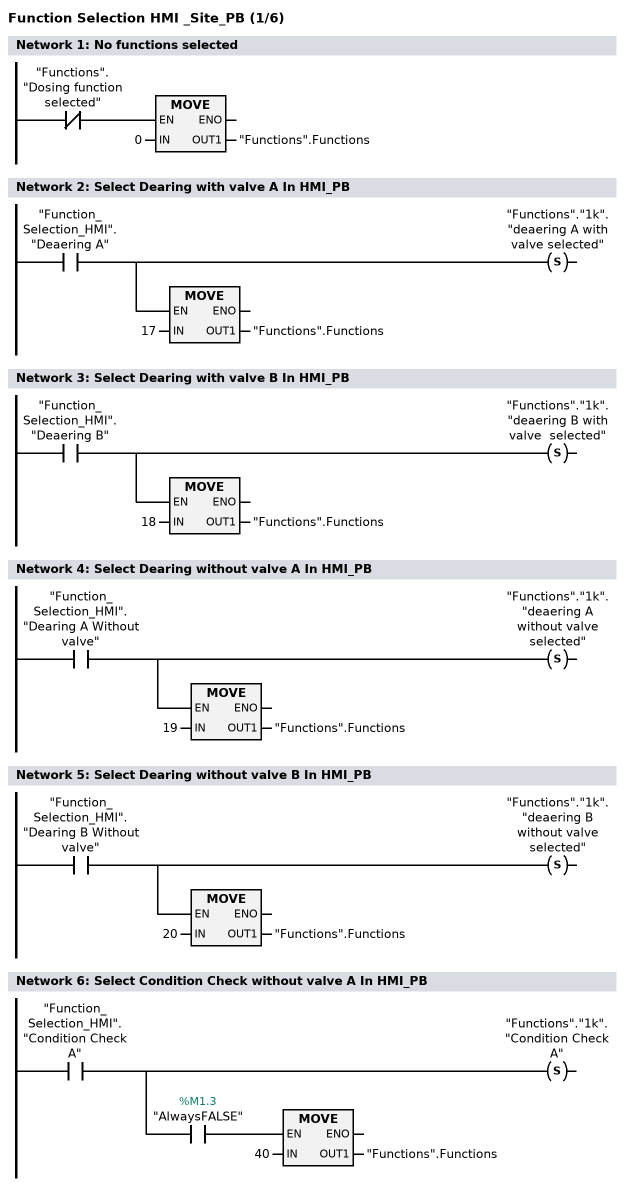
   RUNG wire#powerrail
      I_Contact( "Functions"."Dosing function selected" )
      Move(in := 0, out1 => "Functions".Functions)
   END_RUNG
   // the same network as SCL:
   IF NOT "Functions"."Dosing function selected" THEN "Functions".Functions := 0; END_IF;
END_REGION

REGION Network 2: Select Dearing with valve A In HMI_PB
   RUNG wire#powerrail
      Contact( "Function_Selection_HMI"."Deaering A" )
      wire#w1
      S_Coil( "Functions"."1k"."deaering A with valve selected" )
   END_RUNG
   RUNG wire#w1
      Move(in := 17, out1 => "Functions".Functions)
   END_RUNG
   // the same network as SCL:
   IF "Function_Selection_HMI"."Deaering A" THEN
       "Functions"."1k"."deaering A with valve selected" := TRUE;
       "Functions".Functions := 17;
   END_IF;
END_REGION

REGION Network 3: Select Dearing with valve B In HMI_PB
   RUNG wire#powerrail
      Contact( "Function_Selection_HMI"."Deaering B" )
      wire#w1
      S_Coil( "Functions"."1k"."deaering B with valve  selected" )
   END_RUNG
   RUNG wire#w1
      Move(in := 18, out1 => "Functions".Functions)
   END_RUNG
   // the same network as SCL:
   IF "Function_Selection_HMI"."Deaering B" THEN
       "Functions"."1k"."deaering B with valve  selected" := TRUE;
       "Functions".Functions := 18;
   END_IF;
END_REGION

REGION Network 4: Select Dearing without valve A In HMI_PB
   RUNG wire#powerrail
      Contact( "Function_Selection_HMI"."Dearing A Without valve" )
      wire#w1
      S_Coil( "Functions"."1k"."deaering A without valve selected" )
   END_RUNG
   RUNG wire#w1
      Move(in := 19, out1 => "Functions".Functions)
   END_RUNG
   // the same network as SCL:
   IF "Function_Selection_HMI"."Dearing A Without valve" THEN
       "Functions"."1k"."deaering A without valve selected" := TRUE;
       "Functions".Functions := 19;
   END_IF;
END_REGION

REGION Network 5: Select Dearing without valve B In HMI_PB
   RUNG wire#powerrail
      Contact( "Function_Selection_HMI"."Dearing B Without valve" )
      wire#w1
      S_Coil( "Functions"."1k"."deaering B without valve  selected" )
   END_RUNG
   RUNG wire#w1
      Move(in := 20, out1 => "Functions".Functions)
   END_RUNG
   // the same network as SCL:
   IF "Function_Selection_HMI"."Dearing B Without valve" THEN
       "Functions"."1k"."deaering B without valve  selected" := TRUE;
       "Functions".Functions := 20;
   END_IF;
END_REGION

REGION Network 6: Select Condition Check without valve A In HMI_PB
   RUNG wire#powerrail
      Contact( "Function_Selection_HMI"."Condition Check A" )
      wire#w1
      S_Coil( "Functions"."1k"."Condition Check A" )
   END_RUNG
   RUNG wire#w1
      Contact( "AlwaysFALSE" )
      Move(in := 40, out1 => "Functions".Functions)
   END_RUNG
   // the same network as SCL:
   IF "Function_Selection_HMI"."Condition Check A" THEN "Functions"."1k"."Condition Check A" := TRUE; END_IF;
   IF "Function_Selection_HMI"."Condition Check A" AND "AlwaysFALSE" THEN
       "Functions".Functions := 40;
   END_IF;
END_REGION

REGION Network 7: Select Conditon Check without valve B In HMI_PB
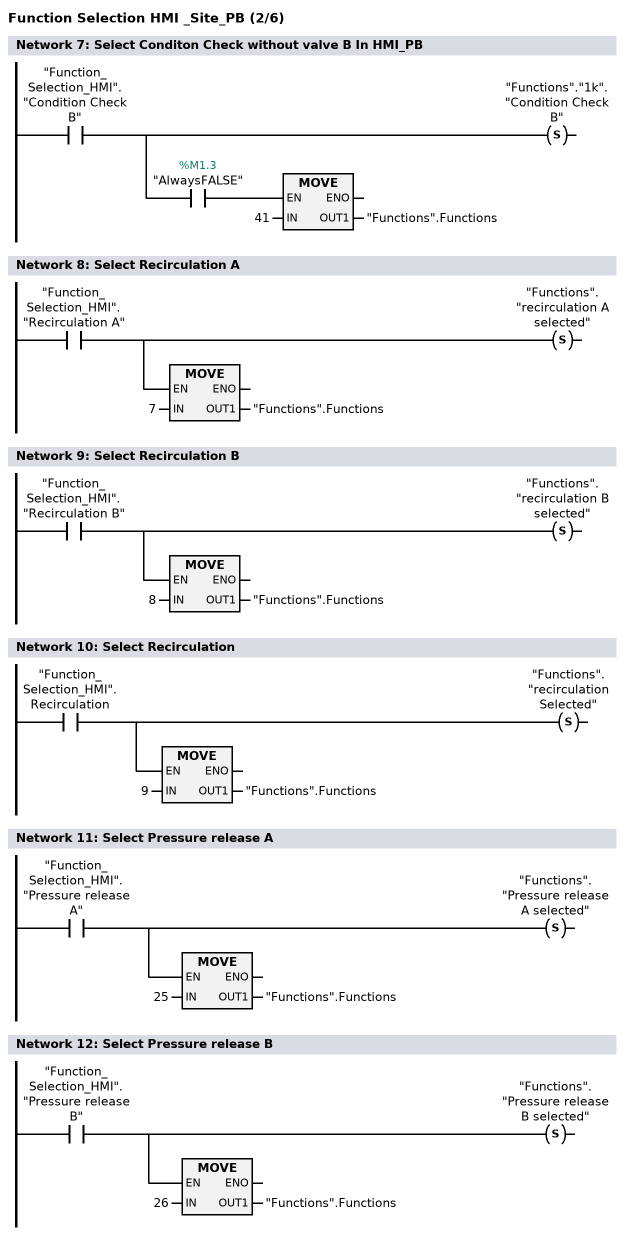
   RUNG wire#powerrail
      Contact( "Function_Selection_HMI"."Condition Check B" )
      wire#w1
      S_Coil( "Functions"."1k"."Condition Check B" )
   END_RUNG
   RUNG wire#w1
      Contact( "AlwaysFALSE" )
      Move(in := 41, out1 => "Functions".Functions)
   END_RUNG
   // the same network as SCL:
   IF "Function_Selection_HMI"."Condition Check B" THEN "Functions"."1k"."Condition Check B" := TRUE; END_IF;
   IF "Function_Selection_HMI"."Condition Check B" AND "AlwaysFALSE" THEN
       "Functions".Functions := 41;
   END_IF;
END_REGION

REGION Network 8: Select Recirculation A
   RUNG wire#powerrail
      Contact( "Function_Selection_HMI"."Recirculation A" )
      wire#w1
      S_Coil( "Functions"."recirculation A selected" )
   END_RUNG
   RUNG wire#w1
      Move(in := 7, out1 => "Functions".Functions)
   END_RUNG
   // the same network as SCL:
   IF "Function_Selection_HMI"."Recirculation A" THEN
       "Functions"."recirculation A selected" := TRUE;
       "Functions".Functions := 7;
   END_IF;
END_REGION

REGION Network 9: Select Recirculation B
   RUNG wire#powerrail
      Contact( "Function_Selection_HMI"."Recirculation B" )
      wire#w1
      S_Coil( "Functions"."recirculation B selected" )
   END_RUNG
   RUNG wire#w1
      Move(in := 8, out1 => "Functions".Functions)
   END_RUNG
   // the same network as SCL:
   IF "Function_Selection_HMI"."Recirculation B" THEN
       "Functions"."recirculation B selected" := TRUE;
       "Functions".Functions := 8;
   END_IF;
END_REGION

REGION Network 10: Select Recirculation
   RUNG wire#powerrail
      Contact( "Function_Selection_HMI".Recirculation )
      wire#w1
      S_Coil( "Functions"."recirculation Selected" )
   END_RUNG
   RUNG wire#w1
      Move(in := 9, out1 => "Functions".Functions)
   END_RUNG
   // the same network as SCL:
   IF "Function_Selection_HMI".Recirculation THEN
       "Functions"."recirculation Selected" := TRUE;
       "Functions".Functions := 9;
   END_IF;
END_REGION

REGION Network 11: Select Pressure release A
   RUNG wire#powerrail
      Contact( "Function_Selection_HMI"."Pressure release A" )
      wire#w1
      S_Coil( "Functions"."Pressure release A selected" )
   END_RUNG
   RUNG wire#w1
      Move(in := 25, out1 => "Functions".Functions)
   END_RUNG
   // the same network as SCL:
   IF "Function_Selection_HMI"."Pressure release A" THEN
       "Functions"."Pressure release A selected" := TRUE;
       "Functions".Functions := 25;
   END_IF;
END_REGION

REGION Network 12: Select Pressure release B
   RUNG wire#powerrail
      Contact( "Function_Selection_HMI"."Pressure release B" )
      wire#w1
      S_Coil( "Functions"."Pressure release B selected" )
   END_RUNG
   RUNG wire#w1
      Move(in := 26, out1 => "Functions".Functions)
   END_RUNG
   // the same network as SCL:
   IF "Function_Selection_HMI"."Pressure release B" THEN
       "Functions"."Pressure release B selected" := TRUE;
       "Functions".Functions := 26;
   END_IF;
END_REGION

REGION Network 13: Select Pressure release
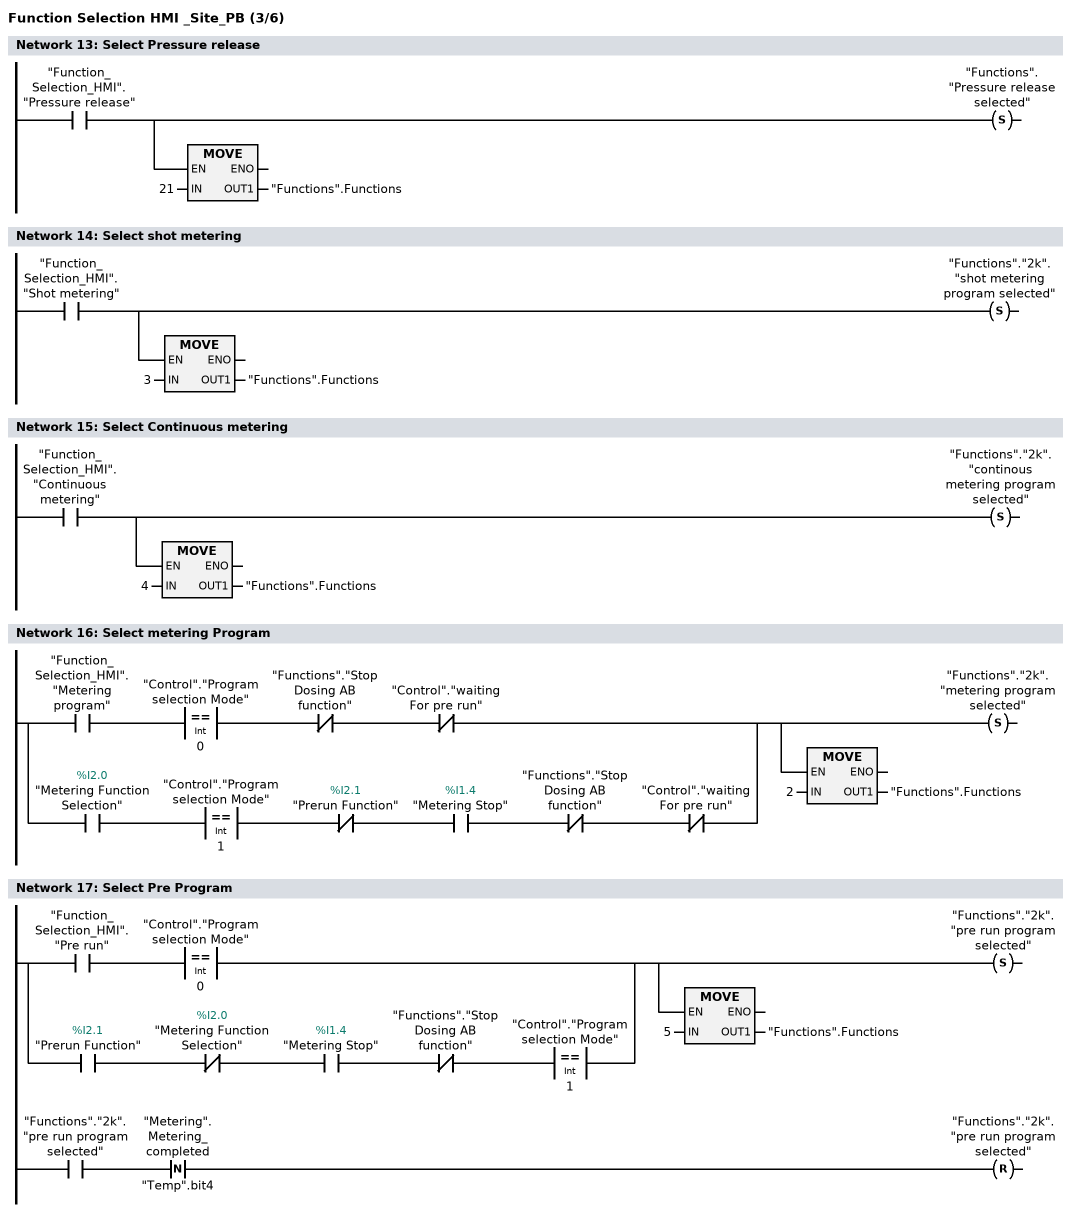
   RUNG wire#powerrail
      Contact( "Function_Selection_HMI"."Pressure release" )
      wire#w1
      S_Coil( "Functions"."Pressure release selected" )
   END_RUNG
   RUNG wire#w1
      Move(in := 21, out1 => "Functions".Functions)
   END_RUNG
   // the same network as SCL:
   IF "Function_Selection_HMI"."Pressure release" THEN
       "Functions"."Pressure release selected" := TRUE;
       "Functions".Functions := 21;
   END_IF;
END_REGION

REGION Network 14: Select shot metering
   RUNG wire#powerrail
      Contact( "Function_Selection_HMI"."Shot metering" )
      wire#w1
      S_Coil( "Functions"."2k"."shot metering program selected" )
   END_RUNG
   RUNG wire#w1
      Move(in := 3, out1 => "Functions".Functions)
   END_RUNG
   // the same network as SCL:
   IF "Function_Selection_HMI"."Shot metering" THEN
       "Functions"."2k"."shot metering program selected" := TRUE;
       "Functions".Functions := 3;
   END_IF;
END_REGION

REGION Network 15: Select Continuous metering
   RUNG wire#powerrail
      Contact( "Function_Selection_HMI"."Continuous metering" )
      wire#w1
      S_Coil( "Functions"."2k"."continous metering program selected" )
   END_RUNG
   RUNG wire#w1
      Move(in := 4, out1 => "Functions".Functions)
   END_RUNG
   // the same network as SCL:
   IF "Function_Selection_HMI"."Continuous metering" THEN
       "Functions"."2k"."continous metering program selected" := TRUE;
       "Functions".Functions := 4;
   END_IF;
END_REGION

REGION Network 16: Select metering Program
   RUNG wire#powerrail
      Contact( "Function_Selection_HMI"."Metering program" )
      { S7_Templates := "SrcType := Int" } EQ_Contact(in1 := "Control"."Program selection Mode", in2 := 0)
      I_Contact( "Functions"."Stop Dosing AB function" )
      I_Contact( "Control"."waiting For pre run" )
      wire#w1
      S_Coil( "Functions"."2k"."metering program selected" )
   END_RUNG
   RUNG wire#powerrail
      Contact( "Metering Function Selection" )
      { S7_Templates := "SrcType := Int" } EQ_Contact(in1 := "Control"."Program selection Mode", in2 := 1)
      I_Contact( "Prerun Function" )
      Contact( "Metering Stop" )
      I_Contact( "Functions"."Stop Dosing AB function" )
      I_Contact( "Control"."waiting For pre run" )
   END_RUNG wire#w1
   RUNG wire#w1
      Move(in := 2, out1 => "Functions".Functions)
   END_RUNG
   // the same network as SCL:
   IF ("Function_Selection_HMI"."Metering program" AND ("Control"."Program selection Mode" = 0) AND NOT "Functions"."Stop Dosing AB function" AND NOT "Control"."waiting For pre run") OR ("Metering Function Selection" AND ("Control"."Program selection Mode" = 1) AND NOT "Prerun Function" AND "Metering Stop" AND NOT "Functions"."Stop Dosing AB function" AND NOT "Control"."waiting For pre run") THEN
       "Functions"."2k"."metering program selected" := TRUE;
       "Functions".Functions := 2;
   END_IF;
END_REGION

REGION Network 17: Select Pre Program
   RUNG wire#powerrail
      Contact( "Function_Selection_HMI"."Pre run" )
      { S7_Templates := "SrcType := Int" } EQ_Contact(in1 := "Control"."Program selection Mode", in2 := 0)
      wire#w1
      S_Coil( "Functions"."2k"."pre run program selected" )
   END_RUNG
   RUNG wire#powerrail
      Contact( "Prerun Function" )
      I_Contact( "Metering Function Selection" )
      Contact( "Metering Stop" )
      I_Contact( "Functions"."Stop Dosing AB function" )
      { S7_Templates := "SrcType := Int" } EQ_Contact(in1 := "Control"."Program selection Mode", in2 := 1)
   END_RUNG wire#w1
   RUNG wire#w1
      Move(in := 5, out1 => "Functions".Functions)
   END_RUNG
   RUNG wire#powerrail
      Contact( "Functions"."2k"."pre run program selected" )
      N_Contact(operand := "Metering".Metering_completed, bit := "Temp".bit4)
      R_Coil( "Functions"."2k"."pre run program selected" )
   END_RUNG
   // the same network as SCL:
   IF ("Function_Selection_HMI"."Pre run" AND ("Control"."Program selection Mode" = 0)) OR ("Prerun Function" AND NOT "Metering Function Selection" AND "Metering Stop" AND NOT "Functions"."Stop Dosing AB function" AND ("Control"."Program selection Mode" = 1)) THEN
       "Functions"."2k"."pre run program selected" := TRUE;
       "Functions".Functions := 5;
   END_IF;
   #_w1 := "Functions"."2k"."pre run program selected" AND NOT "Metering".Metering_completed AND "Temp".bit4;   // falling edge of "Metering".Metering_completed
   "Temp".bit4 := "Metering".Metering_completed;
   IF #_w1 THEN "Functions"."2k"."pre run program selected" := FALSE; END_IF;
END_REGION

REGION Network 18: Select Ratio Program
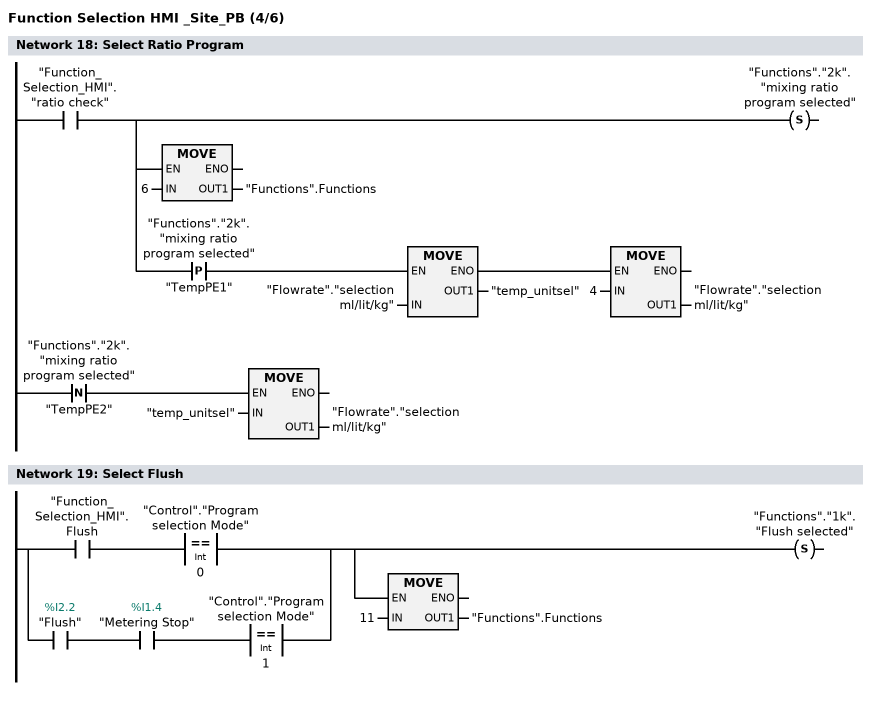
   RUNG wire#powerrail
      Contact( "Function_Selection_HMI"."ratio check" )
      wire#w1
      S_Coil( "Functions"."2k"."mixing ratio program selected" )
   END_RUNG
   RUNG wire#w1
      Move(in := 6, out1 => "Functions".Functions)
   END_RUNG
   RUNG wire#w1
      P_Contact(operand := "Functions"."2k"."mixing ratio program selected", bit := "TempPE1")
      Move(in := "Flowrate"."selection ml/lit/kg", out1 => "temp_unitsel")
      Move(in := 4, out1 => "Flowrate"."selection ml/lit/kg")
   END_RUNG
   RUNG wire#powerrail
      N_Contact(operand := "Functions"."2k"."mixing ratio program selected", bit := "TempPE2")
      Move(in := "temp_unitsel", out1 => "Flowrate"."selection ml/lit/kg")
   END_RUNG
   // the same network as SCL:
   IF "Function_Selection_HMI"."ratio check" THEN
       "Functions"."2k"."mixing ratio program selected" := TRUE;
       "Functions".Functions := 6;
   END_IF;
   #_w1 := "Function_Selection_HMI"."ratio check" AND "Functions"."2k"."mixing ratio program selected" AND NOT "TempPE1";   // rising edge of "Functions"."2k"."mixing ratio program selected"
   "TempPE1" := "Functions"."2k"."mixing ratio program selected";
   IF #_w1 THEN
       "temp_unitsel" := "Flowrate"."selection ml/lit/kg";
       "Flowrate"."selection ml/lit/kg" := 4;
   END_IF;
   #_w2 := NOT "Functions"."2k"."mixing ratio program selected" AND "TempPE2";   // falling edge of "Functions"."2k"."mixing ratio program selected"
   "TempPE2" := "Functions"."2k"."mixing ratio program selected";
   IF #_w2 THEN "Flowrate"."selection ml/lit/kg" := "temp_unitsel"; END_IF;
END_REGION

REGION Network 19: Select Flush
   RUNG wire#powerrail
      Contact( "Function_Selection_HMI".Flush )
      { S7_Templates := "SrcType := Int" } EQ_Contact(in1 := "Control"."Program selection Mode", in2 := 0)
      wire#w1
      S_Coil( "Functions"."1k"."Flush selected" )
   END_RUNG
   RUNG wire#powerrail
      Contact( "Flush" )
      Contact( "Metering Stop" )
      { S7_Templates := "SrcType := Int" } EQ_Contact(in1 := "Control"."Program selection Mode", in2 := 1)
   END_RUNG wire#w1
   RUNG wire#w1
      Move(in := 11, out1 => "Functions".Functions)
   END_RUNG
   // the same network as SCL:
   IF ("Function_Selection_HMI".Flush AND ("Control"."Program selection Mode" = 0)) OR ("Flush" AND "Metering Stop" AND ("Control"."Program selection Mode" = 1)) THEN
       "Functions"."1k"."Flush selected" := TRUE;
       "Functions".Functions := 11;
   END_IF;
END_REGION

REGION Network 20: Select Flush during potlife
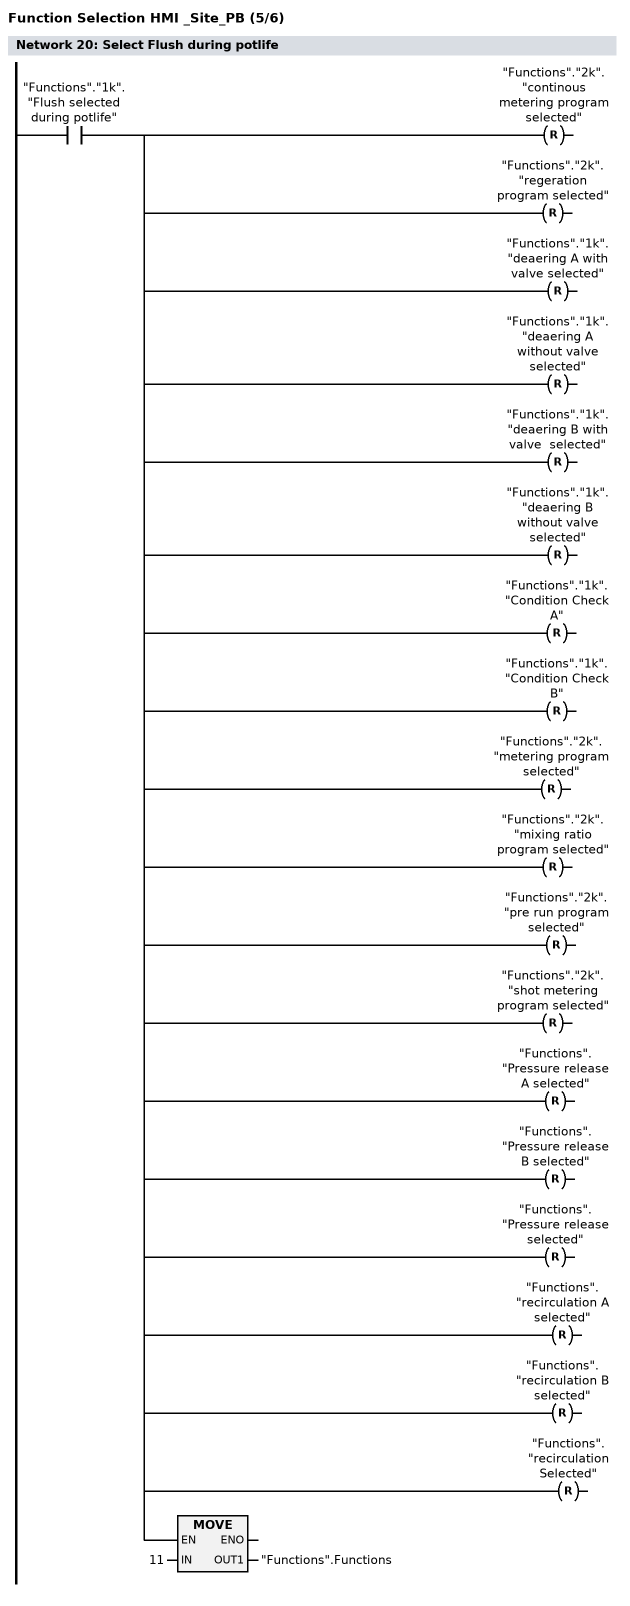
   RUNG wire#powerrail
      Contact( "Functions"."1k"."Flush selected during potlife" )
      wire#w1
      R_Coil( "Functions"."2k"."continous metering program selected" )
   END_RUNG
   RUNG wire#w1
      R_Coil( "Functions"."2k"."regeration program selected" )
   END_RUNG
   RUNG wire#w1
      R_Coil( "Functions"."1k"."deaering A with valve selected" )
   END_RUNG
   RUNG wire#w1
      R_Coil( "Functions"."1k"."deaering A without valve selected" )
   END_RUNG
   RUNG wire#w1
      R_Coil( "Functions"."1k"."deaering B with valve  selected" )
   END_RUNG
   RUNG wire#w1
      R_Coil( "Functions"."1k"."deaering B without valve  selected" )
   END_RUNG
   RUNG wire#w1
      R_Coil( "Functions"."1k"."Condition Check A" )
   END_RUNG
   RUNG wire#w1
      R_Coil( "Functions"."1k"."Condition Check B" )
   END_RUNG
   RUNG wire#w1
      R_Coil( "Functions"."2k"."metering program selected" )
   END_RUNG
   RUNG wire#w1
      R_Coil( "Functions"."2k"."mixing ratio program selected" )
   END_RUNG
   RUNG wire#w1
      R_Coil( "Functions"."2k"."pre run program selected" )
   END_RUNG
   RUNG wire#w1
      R_Coil( "Functions"."2k"."shot metering program selected" )
   END_RUNG
   RUNG wire#w1
      R_Coil( "Functions"."Pressure release A selected" )
   END_RUNG
   RUNG wire#w1
      R_Coil( "Functions"."Pressure release B selected" )
   END_RUNG
   RUNG wire#w1
      R_Coil( "Functions"."Pressure release selected" )
   END_RUNG
   RUNG wire#w1
      R_Coil( "Functions"."recirculation A selected" )
   END_RUNG
   RUNG wire#w1
      R_Coil( "Functions"."recirculation B selected" )
   END_RUNG
   RUNG wire#w1
      R_Coil( "Functions"."recirculation Selected" )
   END_RUNG
   RUNG wire#w1
      Move(in := 11, out1 => "Functions".Functions)
   END_RUNG
   // the same network as SCL:
   IF "Functions"."1k"."Flush selected during potlife" THEN
       "Functions"."2k"."continous metering program selected" := FALSE;
       "Functions"."2k"."regeration program selected" := FALSE;
       "Functions"."1k"."deaering A with valve selected" := FALSE;
       "Functions"."1k"."deaering A without valve selected" := FALSE;
       "Functions"."1k"."deaering B with valve  selected" := FALSE;
       "Functions"."1k"."deaering B without valve  selected" := FALSE;
       "Functions"."1k"."Condition Check A" := FALSE;
       "Functions"."1k"."Condition Check B" := FALSE;
       "Functions"."2k"."metering program selected" := FALSE;
       "Functions"."2k"."mixing ratio program selected" := FALSE;
       "Functions"."2k"."pre run program selected" := FALSE;
       "Functions"."2k"."shot metering program selected" := FALSE;
       "Functions"."Pressure release A selected" := FALSE;
       "Functions"."Pressure release B selected" := FALSE;
       "Functions"."Pressure release selected" := FALSE;
       "Functions"."recirculation A selected" := FALSE;
       "Functions"."recirculation B selected" := FALSE;
       "Functions"."recirculation Selected" := FALSE;
       "Functions".Functions := 11;
   END_IF;
END_REGION

REGION Network 21: regeneration selected
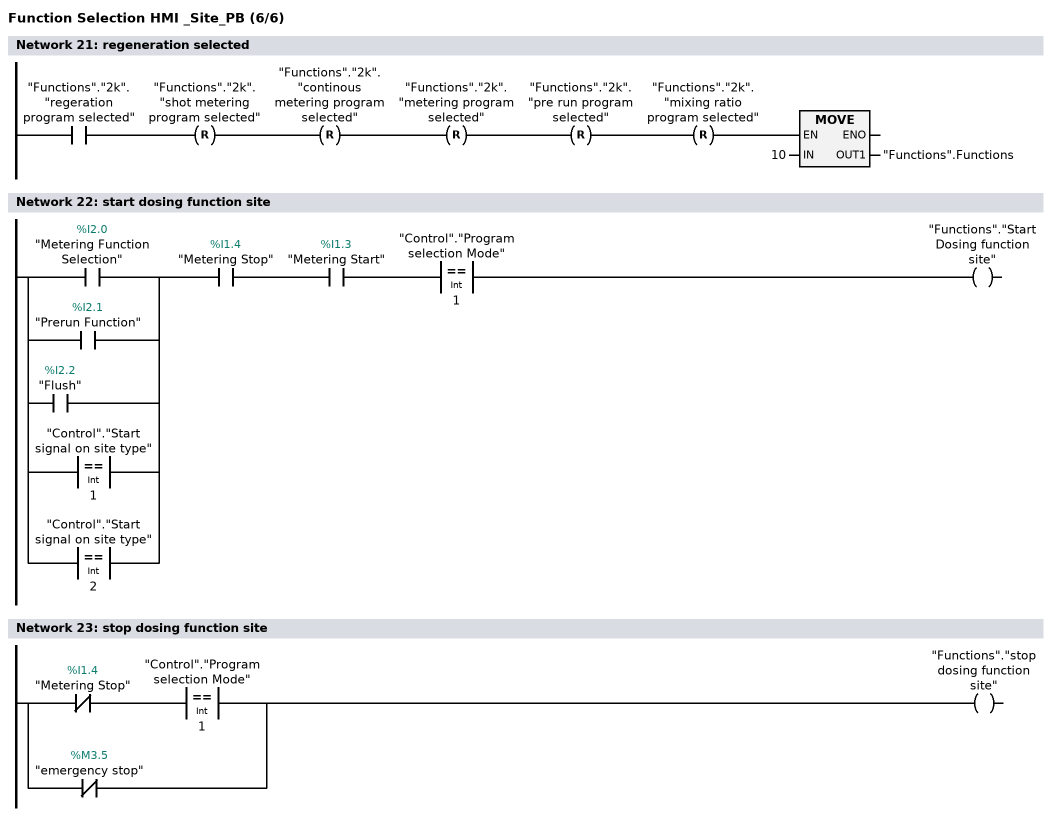
   RUNG wire#powerrail
      Contact( "Functions"."2k"."regeration program selected" )
      R_Coil( "Functions"."2k"."shot metering program selected" )
      R_Coil( "Functions"."2k"."continous metering program selected" )
      R_Coil( "Functions"."2k"."metering program selected" )
      R_Coil( "Functions"."2k"."pre run program selected" )
      R_Coil( "Functions"."2k"."mixing ratio program selected" )
      Move(in := 10, out1 => "Functions".Functions)
   END_RUNG
   // the same network as SCL:
   IF "Functions"."2k"."regeration program selected" THEN
       "Functions"."2k"."shot metering program selected" := FALSE;
       "Functions"."2k"."continous metering program selected" := FALSE;
       "Functions"."2k"."metering program selected" := FALSE;
       "Functions"."2k"."pre run program selected" := FALSE;
       "Functions"."2k"."mixing ratio program selected" := FALSE;
       "Functions".Functions := 10;
   END_IF;
END_REGION

REGION Network 22: start dosing function site
   RUNG wire#powerrail
      Contact( "Metering Function Selection" )
      wire#w1
      Contact( "Metering Stop" )
      Contact( "Metering Start" )
      { S7_Templates := "SrcType := Int" } EQ_Contact(in1 := "Control"."Program selection Mode", in2 := 1)
      Coil( "Functions"."Start Dosing function site" )
   END_RUNG
   RUNG wire#powerrail
      Contact( "Prerun Function" )
   END_RUNG wire#w1
   RUNG wire#powerrail
      Contact( "Flush" )
   END_RUNG wire#w1
   RUNG wire#powerrail
      { S7_Templates := "SrcType := Int" } EQ_Contact(in1 := "Control"."Start signal on site type", in2 := 1)
   END_RUNG wire#w1
   RUNG wire#powerrail
      { S7_Templates := "SrcType := Int" } EQ_Contact(in1 := "Control"."Start signal on site type", in2 := 2)
   END_RUNG wire#w1
   // the same network as SCL:
   "Functions"."Start Dosing function site" := ("Metering Function Selection" OR "Prerun Function" OR "Flush" OR ("Control"."Start signal on site type" = 1) OR ("Control"."Start signal on site type" = 2)) AND "Metering Stop" AND "Metering Start" AND ("Control"."Program selection Mode" = 1);
END_REGION

REGION Network 23: stop dosing function site
   RUNG wire#powerrail
      I_Contact( "Metering Stop" )
      { S7_Templates := "SrcType := Int" } EQ_Contact(in1 := "Control"."Program selection Mode", in2 := 1)
      wire#w1
      Coil( "Functions"."stop dosing function site" )
   END_RUNG
   RUNG wire#powerrail
      I_Contact( "emergency stop" )
   END_RUNG wire#w1
   // the same network as SCL:
   "Functions"."stop dosing function site" := (NOT "Metering Stop" AND ("Control"."Program selection Mode" = 1)) OR NOT "emergency stop";
END_REGION
END_FUNCTION

FUNCTION "HMI screen" : Void   // FC18, LAD
{ S7_Optimized_Access := 'TRUE' }
VERSION : 0.1
// stored: AutoNumber true, IsIECCheckEnabled false, SetENOAutomatically false, UDAEnableTagReadback false
   VAR_TEMP
      temp1 : Bool;
      temp2 : Bool;
      temp3 : Bool;
      temp10 : Bool;
      temp11 : Bool;
      "dearing A" : Bool;
      "dearing A_1" : Bool;
      dearingA : Bool;
   END_VAR
   VAR_TEMP   // added for the SCL form of the ladder/FBD networks
      _w1 : Bool;
      _w2 : Bool;
   END_VAR
BEGIN

REGION Network 1: Metering continious screen/AD1000
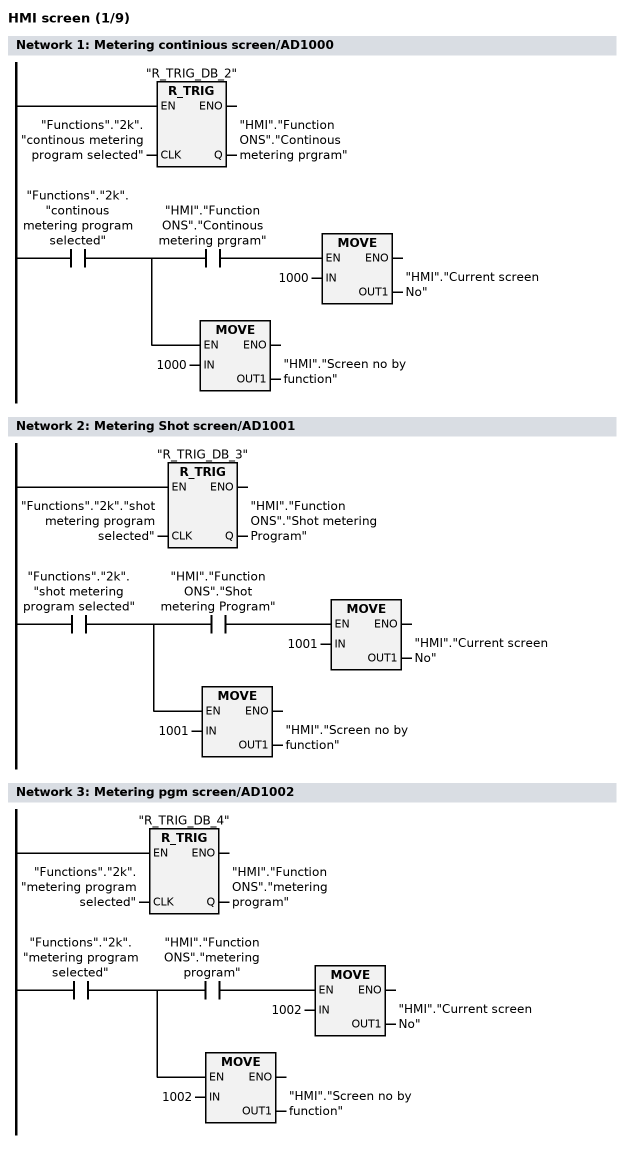
   RUNG wire#powerrail
      "R_TRIG_DB_2".R_TRIG(CLK := "Functions"."2k"."continous metering program selected", Q => "HMI"."Function ONS"."Continous metering prgram")
   END_RUNG
   RUNG wire#powerrail
      Contact( "Functions"."2k"."continous metering program selected" )
      wire#w1
      Contact( "HMI"."Function ONS"."Continous metering prgram" )
      Move(in := 1000, out1 => "HMI"."Current screen No")
   END_RUNG
   RUNG wire#w1
      Move(in := 1000, out1 => "HMI"."Screen no by function")
   END_RUNG
   // the same network as SCL:
   "R_TRIG_DB_2"(CLK := "Functions"."2k"."continous metering program selected",   // R_TRIG
                 Q => "HMI"."Function ONS"."Continous metering prgram");
   IF "Functions"."2k"."continous metering program selected" AND "HMI"."Function ONS"."Continous metering prgram" THEN
       "HMI"."Current screen No" := 1000;
   END_IF;
   IF "Functions"."2k"."continous metering program selected" THEN
       "HMI"."Screen no by function" := 1000;
   END_IF;
END_REGION

REGION Network 2: Metering Shot screen/AD1001
   RUNG wire#powerrail
      "R_TRIG_DB_3".R_TRIG(CLK := "Functions"."2k"."shot metering program selected", Q => "HMI"."Function ONS"."Shot metering Program")
   END_RUNG
   RUNG wire#powerrail
      Contact( "Functions"."2k"."shot metering program selected" )
      wire#w1
      Contact( "HMI"."Function ONS"."Shot metering Program" )
      Move(in := 1001, out1 => "HMI"."Current screen No")
   END_RUNG
   RUNG wire#w1
      Move(in := 1001, out1 => "HMI"."Screen no by function")
   END_RUNG
   // the same network as SCL:
   "R_TRIG_DB_3"(CLK := "Functions"."2k"."shot metering program selected",   // R_TRIG
                 Q => "HMI"."Function ONS"."Shot metering Program");
   IF "Functions"."2k"."shot metering program selected" AND "HMI"."Function ONS"."Shot metering Program" THEN
       "HMI"."Current screen No" := 1001;
   END_IF;
   IF "Functions"."2k"."shot metering program selected" THEN "HMI"."Screen no by function" := 1001; END_IF;
END_REGION

REGION Network 3: Metering pgm screen/AD1002
   RUNG wire#powerrail
      "R_TRIG_DB_4".R_TRIG(CLK := "Functions"."2k"."metering program selected", Q => "HMI"."Function ONS"."metering program")
   END_RUNG
   RUNG wire#powerrail
      Contact( "Functions"."2k"."metering program selected" )
      wire#w1
      Contact( "HMI"."Function ONS"."metering program" )
      Move(in := 1002, out1 => "HMI"."Current screen No")
   END_RUNG
   RUNG wire#w1
      Move(in := 1002, out1 => "HMI"."Screen no by function")
   END_RUNG
   // the same network as SCL:
   "R_TRIG_DB_4"(CLK := "Functions"."2k"."metering program selected",   // R_TRIG
                 Q => "HMI"."Function ONS"."metering program");
   IF "Functions"."2k"."metering program selected" AND "HMI"."Function ONS"."metering program" THEN
       "HMI"."Current screen No" := 1002;
   END_IF;
   IF "Functions"."2k"."metering program selected" THEN "HMI"."Screen no by function" := 1002; END_IF;
END_REGION

REGION Network 4: pre run screen/AD1003
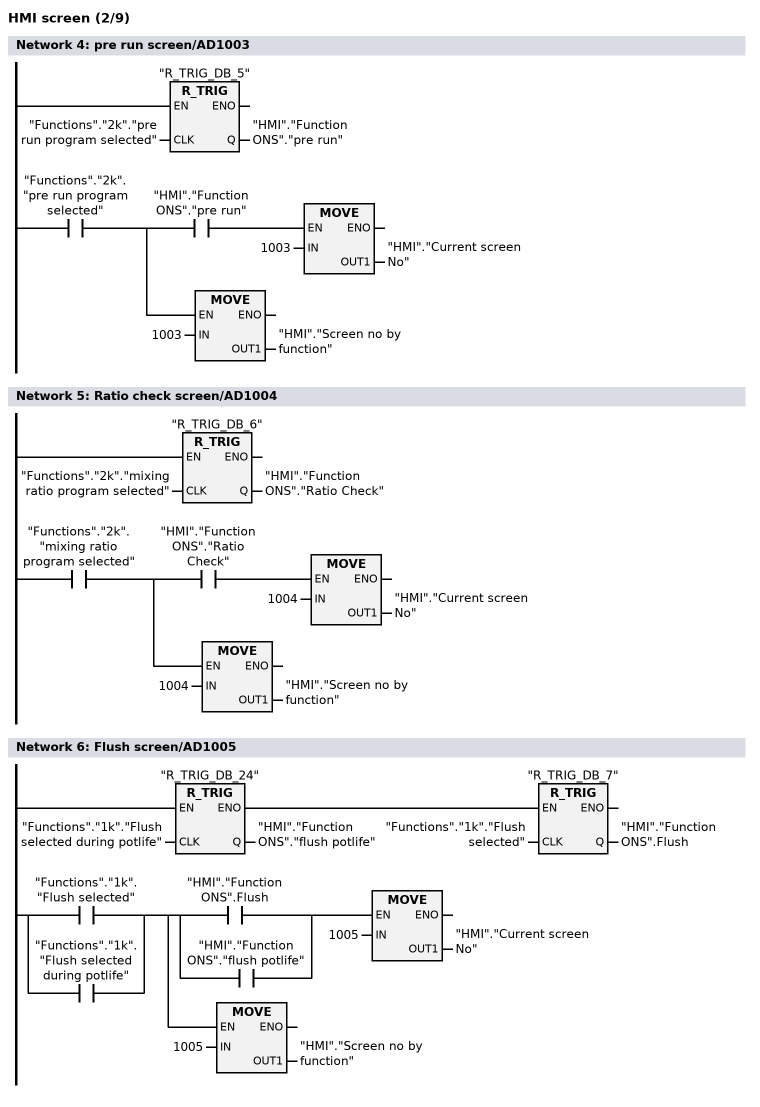
   RUNG wire#powerrail
      "R_TRIG_DB_5".R_TRIG(CLK := "Functions"."2k"."pre run program selected", Q => "HMI"."Function ONS"."pre run")
   END_RUNG
   RUNG wire#powerrail
      Contact( "Functions"."2k"."pre run program selected" )
      wire#w1
      Contact( "HMI"."Function ONS"."pre run" )
      Move(in := 1003, out1 => "HMI"."Current screen No")
   END_RUNG
   RUNG wire#w1
      Move(in := 1003, out1 => "HMI"."Screen no by function")
   END_RUNG
   // the same network as SCL:
   "R_TRIG_DB_5"(CLK := "Functions"."2k"."pre run program selected", Q => "HMI"."Function ONS"."pre run");   // R_TRIG
   IF "Functions"."2k"."pre run program selected" AND "HMI"."Function ONS"."pre run" THEN
       "HMI"."Current screen No" := 1003;
   END_IF;
   IF "Functions"."2k"."pre run program selected" THEN "HMI"."Screen no by function" := 1003; END_IF;
END_REGION

REGION Network 5: Ratio check screen/AD1004
   RUNG wire#powerrail
      "R_TRIG_DB_6".R_TRIG(CLK := "Functions"."2k"."mixing ratio program selected", Q => "HMI"."Function ONS"."Ratio Check")
   END_RUNG
   RUNG wire#powerrail
      Contact( "Functions"."2k"."mixing ratio program selected" )
      wire#w1
      Contact( "HMI"."Function ONS"."Ratio Check" )
      Move(in := 1004, out1 => "HMI"."Current screen No")
   END_RUNG
   RUNG wire#w1
      Move(in := 1004, out1 => "HMI"."Screen no by function")
   END_RUNG
   // the same network as SCL:
   "R_TRIG_DB_6"(CLK := "Functions"."2k"."mixing ratio program selected",   // R_TRIG
                 Q => "HMI"."Function ONS"."Ratio Check");
   IF "Functions"."2k"."mixing ratio program selected" AND "HMI"."Function ONS"."Ratio Check" THEN
       "HMI"."Current screen No" := 1004;
   END_IF;
   IF "Functions"."2k"."mixing ratio program selected" THEN "HMI"."Screen no by function" := 1004; END_IF;
END_REGION

REGION Network 6: Flush screen/AD1005
   RUNG wire#powerrail
      "R_TRIG_DB_24".R_TRIG(CLK := "Functions"."1k"."Flush selected during potlife", Q => "HMI"."Function ONS"."flush potlife")
      "R_TRIG_DB_7".R_TRIG(CLK := "Functions"."1k"."Flush selected", Q => "HMI"."Function ONS".Flush)
   END_RUNG
   RUNG wire#powerrail
      Contact( "Functions"."1k"."Flush selected" )
      wire#w1
      Contact( "HMI"."Function ONS".Flush )
      wire#w2
      Move(in := 1005, out1 => "HMI"."Current screen No")
   END_RUNG
   RUNG wire#powerrail
      Contact( "Functions"."1k"."Flush selected during potlife" )
   END_RUNG wire#w1
   RUNG wire#w1
      Contact( "HMI"."Function ONS"."flush potlife" )
   END_RUNG wire#w2
   RUNG wire#w1
      Move(in := 1005, out1 => "HMI"."Screen no by function")
   END_RUNG
   // the same network as SCL:
   "R_TRIG_DB_24"(CLK := "Functions"."1k"."Flush selected during potlife",   // R_TRIG
                  Q => "HMI"."Function ONS"."flush potlife",
                  ENO => #_w1);
   IF #_w1 THEN
       "R_TRIG_DB_7"(CLK := "Functions"."1k"."Flush selected", Q => "HMI"."Function ONS".Flush);   // R_TRIG
   END_IF;
   #_w2 := "Functions"."1k"."Flush selected" OR "Functions"."1k"."Flush selected during potlife";
   IF #_w2 AND ("HMI"."Function ONS".Flush OR "HMI"."Function ONS"."flush potlife") THEN
       "HMI"."Current screen No" := 1005;
   END_IF;
   IF #_w2 THEN "HMI"."Screen no by function" := 1005; END_IF;
END_REGION

REGION Network 7: dearing A screen/AD1006
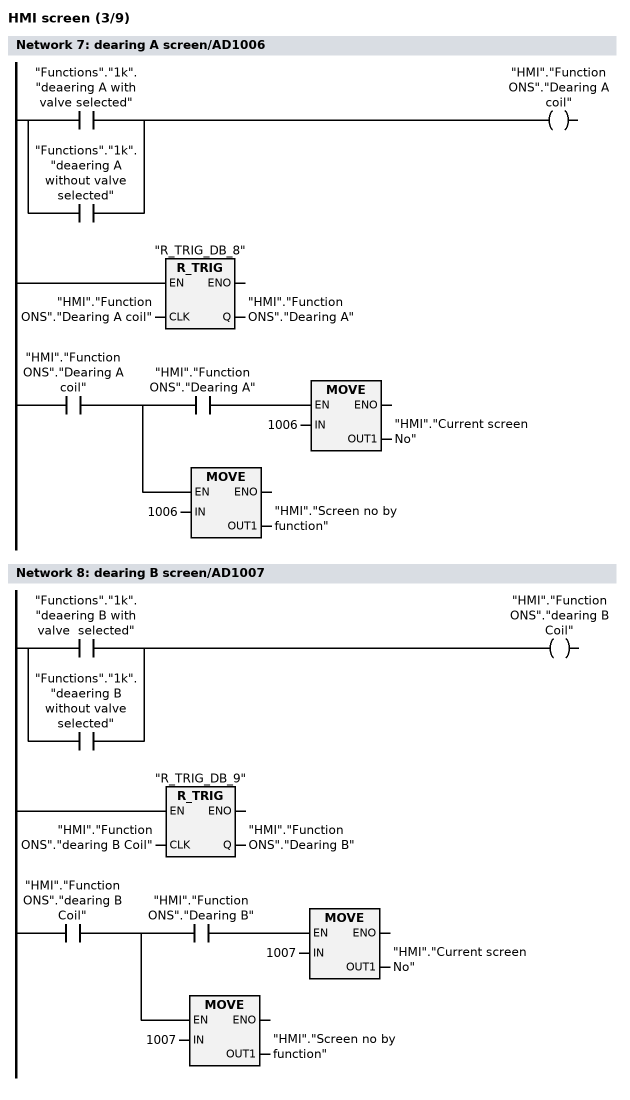
   RUNG wire#powerrail
      Contact( "Functions"."1k"."deaering A with valve selected" )
      wire#w1
      Coil( "HMI"."Function ONS"."Dearing A coil" )
   END_RUNG
   RUNG wire#powerrail
      Contact( "Functions"."1k"."deaering A without valve selected" )
   END_RUNG wire#w1
   RUNG wire#powerrail
      "R_TRIG_DB_8".R_TRIG(CLK := "HMI"."Function ONS"."Dearing A coil", Q => "HMI"."Function ONS"."Dearing A")
   END_RUNG
   RUNG wire#powerrail
      Contact( "HMI"."Function ONS"."Dearing A coil" )
      wire#w2
      Contact( "HMI"."Function ONS"."Dearing A" )
      Move(in := 1006, out1 => "HMI"."Current screen No")
   END_RUNG
   RUNG wire#w2
      Move(in := 1006, out1 => "HMI"."Screen no by function")
   END_RUNG
   // the same network as SCL:
   "HMI"."Function ONS"."Dearing A coil" := "Functions"."1k"."deaering A with valve selected" OR "Functions"."1k"."deaering A without valve selected";
   "R_TRIG_DB_8"(CLK := "HMI"."Function ONS"."Dearing A coil", Q => "HMI"."Function ONS"."Dearing A");   // R_TRIG
   IF "HMI"."Function ONS"."Dearing A coil" AND "HMI"."Function ONS"."Dearing A" THEN
       "HMI"."Current screen No" := 1006;
   END_IF;
   IF "HMI"."Function ONS"."Dearing A coil" THEN "HMI"."Screen no by function" := 1006; END_IF;
END_REGION

REGION Network 8: dearing B screen/AD1007
   RUNG wire#powerrail
      Contact( "Functions"."1k"."deaering B with valve  selected" )
      wire#w1
      Coil( "HMI"."Function ONS"."dearing B Coil" )
   END_RUNG
   RUNG wire#powerrail
      Contact( "Functions"."1k"."deaering B without valve  selected" )
   END_RUNG wire#w1
   RUNG wire#powerrail
      "R_TRIG_DB_9".R_TRIG(CLK := "HMI"."Function ONS"."dearing B Coil", Q => "HMI"."Function ONS"."Dearing B")
   END_RUNG
   RUNG wire#powerrail
      Contact( "HMI"."Function ONS"."dearing B Coil" )
      wire#w2
      Contact( "HMI"."Function ONS"."Dearing B" )
      Move(in := 1007, out1 => "HMI"."Current screen No")
   END_RUNG
   RUNG wire#w2
      Move(in := 1007, out1 => "HMI"."Screen no by function")
   END_RUNG
   // the same network as SCL:
   "HMI"."Function ONS"."dearing B Coil" := "Functions"."1k"."deaering B with valve  selected" OR "Functions"."1k"."deaering B without valve  selected";
   "R_TRIG_DB_9"(CLK := "HMI"."Function ONS"."dearing B Coil", Q => "HMI"."Function ONS"."Dearing B");   // R_TRIG
   IF "HMI"."Function ONS"."dearing B Coil" AND "HMI"."Function ONS"."Dearing B" THEN
       "HMI"."Current screen No" := 1007;
   END_IF;
   IF "HMI"."Function ONS"."dearing B Coil" THEN "HMI"."Screen no by function" := 1007; END_IF;
END_REGION

REGION Network 9: Condition Check A screen/AD1015
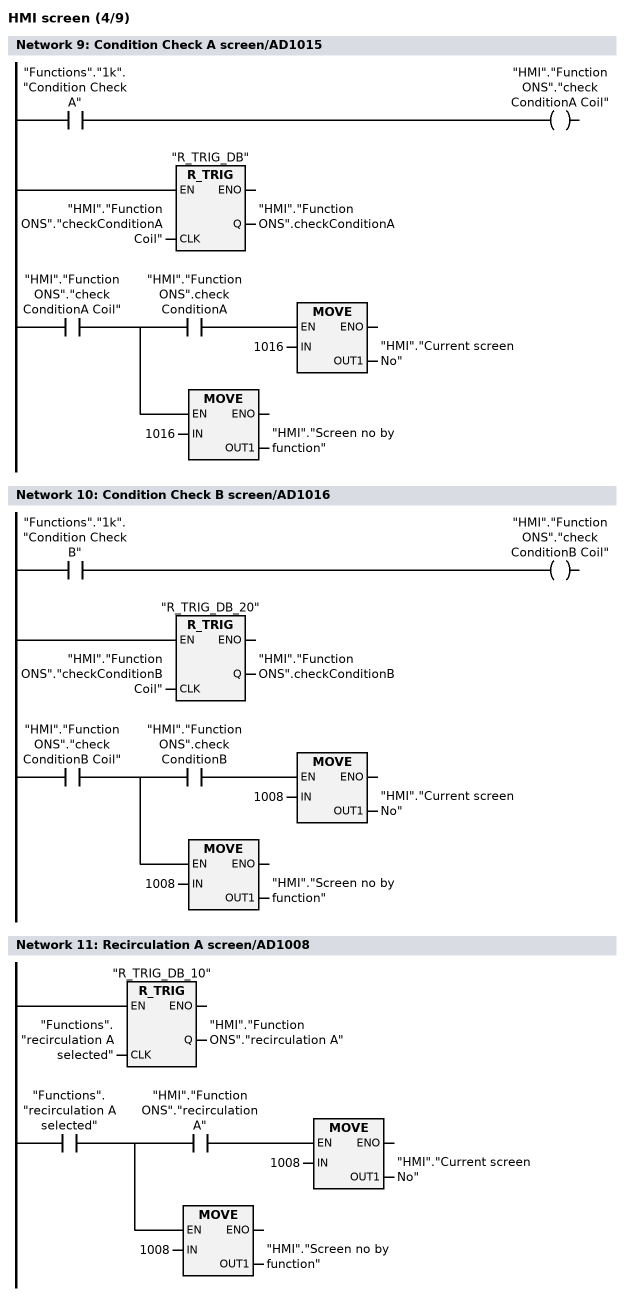
   RUNG wire#powerrail
      Contact( "Functions"."1k"."Condition Check A" )
      Coil( "HMI"."Function ONS"."checkConditionA Coil" )
   END_RUNG
   RUNG wire#powerrail
      "R_TRIG_DB".R_TRIG(CLK := "HMI"."Function ONS"."checkConditionA Coil", Q => "HMI"."Function ONS".checkConditionA)
   END_RUNG
   RUNG wire#powerrail
      Contact( "HMI"."Function ONS"."checkConditionA Coil" )
      wire#w1
      Contact( "HMI"."Function ONS".checkConditionA )
      Move(in := 1016, out1 => "HMI"."Current screen No")
   END_RUNG
   RUNG wire#w1
      Move(in := 1016, out1 => "HMI"."Screen no by function")
   END_RUNG
   // the same network as SCL:
   "HMI"."Function ONS"."checkConditionA Coil" := "Functions"."1k"."Condition Check A";
   "R_TRIG_DB"(CLK := "HMI"."Function ONS"."checkConditionA Coil", Q => "HMI"."Function ONS".checkConditionA);   // R_TRIG
   IF "HMI"."Function ONS"."checkConditionA Coil" AND "HMI"."Function ONS".checkConditionA THEN
       "HMI"."Current screen No" := 1016;
   END_IF;
   IF "HMI"."Function ONS"."checkConditionA Coil" THEN "HMI"."Screen no by function" := 1016; END_IF;
END_REGION

REGION Network 10: Condition Check B screen/AD1016
   RUNG wire#powerrail
      Contact( "Functions"."1k"."Condition Check B" )
      Coil( "HMI"."Function ONS"."checkConditionB Coil" )
   END_RUNG
   RUNG wire#powerrail
      "R_TRIG_DB_20".R_TRIG(CLK := "HMI"."Function ONS"."checkConditionB Coil", Q => "HMI"."Function ONS".checkConditionB)
   END_RUNG
   RUNG wire#powerrail
      Contact( "HMI"."Function ONS"."checkConditionB Coil" )
      wire#w1
      Contact( "HMI"."Function ONS".checkConditionB )
      Move(in := 1008, out1 => "HMI"."Current screen No")
   END_RUNG
   RUNG wire#w1
      Move(in := 1008, out1 => "HMI"."Screen no by function")
   END_RUNG
   // the same network as SCL:
   "HMI"."Function ONS"."checkConditionB Coil" := "Functions"."1k"."Condition Check B";
   "R_TRIG_DB_20"(CLK := "HMI"."Function ONS"."checkConditionB Coil", Q => "HMI"."Function ONS".checkConditionB);   // R_TRIG
   IF "HMI"."Function ONS"."checkConditionB Coil" AND "HMI"."Function ONS".checkConditionB THEN
       "HMI"."Current screen No" := 1008;
   END_IF;
   IF "HMI"."Function ONS"."checkConditionB Coil" THEN "HMI"."Screen no by function" := 1008; END_IF;
END_REGION

REGION Network 11: Recirculation A screen/AD1008
   RUNG wire#powerrail
      "R_TRIG_DB_10".R_TRIG(CLK := "Functions"."recirculation A selected", Q => "HMI"."Function ONS"."recirculation A")
   END_RUNG
   RUNG wire#powerrail
      Contact( "Functions"."recirculation A selected" )
      wire#w1
      Contact( "HMI"."Function ONS"."recirculation A" )
      Move(in := 1008, out1 => "HMI"."Current screen No")
   END_RUNG
   RUNG wire#w1
      Move(in := 1008, out1 => "HMI"."Screen no by function")
   END_RUNG
   // the same network as SCL:
   "R_TRIG_DB_10"(CLK := "Functions"."recirculation A selected", Q => "HMI"."Function ONS"."recirculation A");   // R_TRIG
   IF "Functions"."recirculation A selected" AND "HMI"."Function ONS"."recirculation A" THEN
       "HMI"."Current screen No" := 1008;
   END_IF;
   IF "Functions"."recirculation A selected" THEN "HMI"."Screen no by function" := 1008; END_IF;
END_REGION

REGION Network 12: Recirculation B screen/AD1009
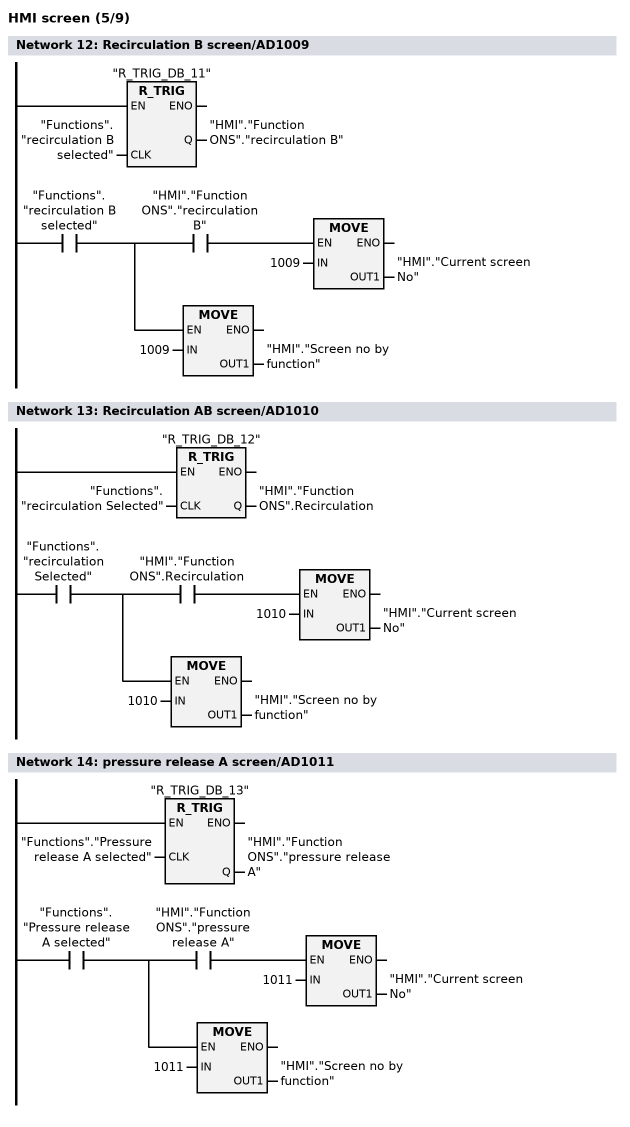
   RUNG wire#powerrail
      "R_TRIG_DB_11".R_TRIG(CLK := "Functions"."recirculation B selected", Q => "HMI"."Function ONS"."recirculation B")
   END_RUNG
   RUNG wire#powerrail
      Contact( "Functions"."recirculation B selected" )
      wire#w1
      Contact( "HMI"."Function ONS"."recirculation B" )
      Move(in := 1009, out1 => "HMI"."Current screen No")
   END_RUNG
   RUNG wire#w1
      Move(in := 1009, out1 => "HMI"."Screen no by function")
   END_RUNG
   // the same network as SCL:
   "R_TRIG_DB_11"(CLK := "Functions"."recirculation B selected", Q => "HMI"."Function ONS"."recirculation B");   // R_TRIG
   IF "Functions"."recirculation B selected" AND "HMI"."Function ONS"."recirculation B" THEN
       "HMI"."Current screen No" := 1009;
   END_IF;
   IF "Functions"."recirculation B selected" THEN "HMI"."Screen no by function" := 1009; END_IF;
END_REGION

REGION Network 13: Recirculation AB screen/AD1010
   RUNG wire#powerrail
      "R_TRIG_DB_12".R_TRIG(CLK := "Functions"."recirculation Selected", Q => "HMI"."Function ONS".Recirculation)
   END_RUNG
   RUNG wire#powerrail
      Contact( "Functions"."recirculation Selected" )
      wire#w1
      Contact( "HMI"."Function ONS".Recirculation )
      Move(in := 1010, out1 => "HMI"."Current screen No")
   END_RUNG
   RUNG wire#w1
      Move(in := 1010, out1 => "HMI"."Screen no by function")
   END_RUNG
   // the same network as SCL:
   "R_TRIG_DB_12"(CLK := "Functions"."recirculation Selected", Q => "HMI"."Function ONS".Recirculation);   // R_TRIG
   IF "Functions"."recirculation Selected" AND "HMI"."Function ONS".Recirculation THEN
       "HMI"."Current screen No" := 1010;
   END_IF;
   IF "Functions"."recirculation Selected" THEN "HMI"."Screen no by function" := 1010; END_IF;
END_REGION

REGION Network 14: pressure release A screen/AD1011
   RUNG wire#powerrail
      "R_TRIG_DB_13".R_TRIG(CLK := "Functions"."Pressure release A selected", Q => "HMI"."Function ONS"."pressure release A")
   END_RUNG
   RUNG wire#powerrail
      Contact( "Functions"."Pressure release A selected" )
      wire#w1
      Contact( "HMI"."Function ONS"."pressure release A" )
      Move(in := 1011, out1 => "HMI"."Current screen No")
   END_RUNG
   RUNG wire#w1
      Move(in := 1011, out1 => "HMI"."Screen no by function")
   END_RUNG
   // the same network as SCL:
   "R_TRIG_DB_13"(CLK := "Functions"."Pressure release A selected",   // R_TRIG
                  Q => "HMI"."Function ONS"."pressure release A");
   IF "Functions"."Pressure release A selected" AND "HMI"."Function ONS"."pressure release A" THEN
       "HMI"."Current screen No" := 1011;
   END_IF;
   IF "Functions"."Pressure release A selected" THEN "HMI"."Screen no by function" := 1011; END_IF;
END_REGION

REGION Network 15: pressure release B screen/AD1012
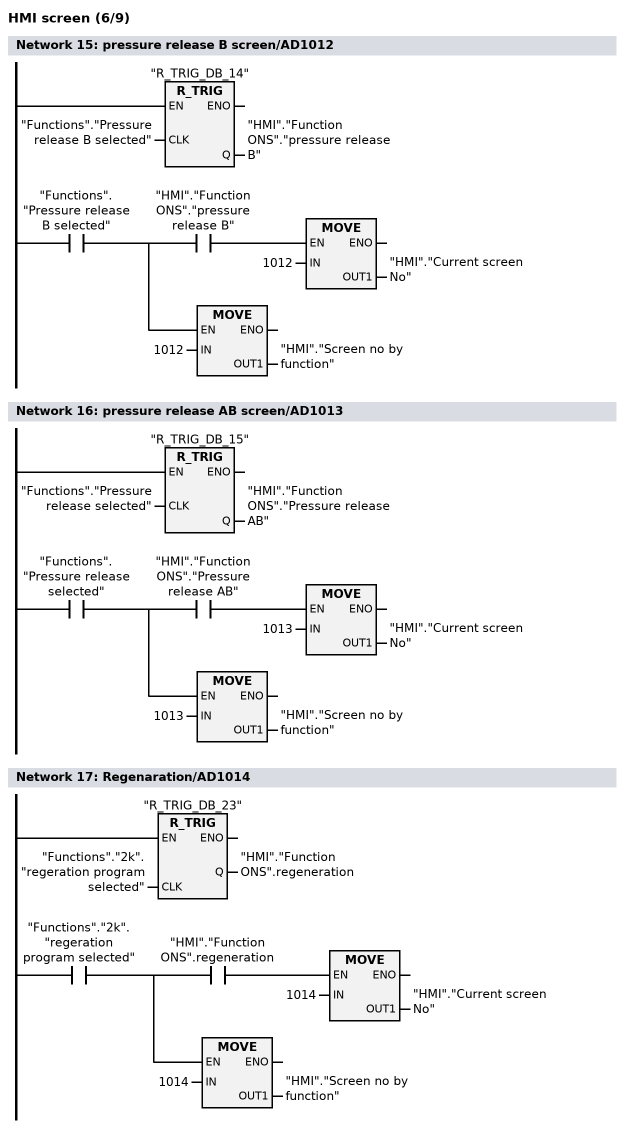
   RUNG wire#powerrail
      "R_TRIG_DB_14".R_TRIG(CLK := "Functions"."Pressure release B selected", Q => "HMI"."Function ONS"."pressure release B")
   END_RUNG
   RUNG wire#powerrail
      Contact( "Functions"."Pressure release B selected" )
      wire#w1
      Contact( "HMI"."Function ONS"."pressure release B" )
      Move(in := 1012, out1 => "HMI"."Current screen No")
   END_RUNG
   RUNG wire#w1
      Move(in := 1012, out1 => "HMI"."Screen no by function")
   END_RUNG
   // the same network as SCL:
   "R_TRIG_DB_14"(CLK := "Functions"."Pressure release B selected",   // R_TRIG
                  Q => "HMI"."Function ONS"."pressure release B");
   IF "Functions"."Pressure release B selected" AND "HMI"."Function ONS"."pressure release B" THEN
       "HMI"."Current screen No" := 1012;
   END_IF;
   IF "Functions"."Pressure release B selected" THEN "HMI"."Screen no by function" := 1012; END_IF;
END_REGION

REGION Network 16: pressure release AB screen/AD1013
   RUNG wire#powerrail
      "R_TRIG_DB_15".R_TRIG(CLK := "Functions"."Pressure release selected", Q => "HMI"."Function ONS"."Pressure release AB")
   END_RUNG
   RUNG wire#powerrail
      Contact( "Functions"."Pressure release selected" )
      wire#w1
      Contact( "HMI"."Function ONS"."Pressure release AB" )
      Move(in := 1013, out1 => "HMI"."Current screen No")
   END_RUNG
   RUNG wire#w1
      Move(in := 1013, out1 => "HMI"."Screen no by function")
   END_RUNG
   // the same network as SCL:
   "R_TRIG_DB_15"(CLK := "Functions"."Pressure release selected",   // R_TRIG
                  Q => "HMI"."Function ONS"."Pressure release AB");
   IF "Functions"."Pressure release selected" AND "HMI"."Function ONS"."Pressure release AB" THEN
       "HMI"."Current screen No" := 1013;
   END_IF;
   IF "Functions"."Pressure release selected" THEN "HMI"."Screen no by function" := 1013; END_IF;
END_REGION

REGION Network 17: Regenaration/AD1014
   RUNG wire#powerrail
      "R_TRIG_DB_23".R_TRIG(CLK := "Functions"."2k"."regeration program selected", Q => "HMI"."Function ONS".regeneration)
   END_RUNG
   RUNG wire#powerrail
      Contact( "Functions"."2k"."regeration program selected" )
      wire#w1
      Contact( "HMI"."Function ONS".regeneration )
      Move(in := 1014, out1 => "HMI"."Current screen No")
   END_RUNG
   RUNG wire#w1
      Move(in := 1014, out1 => "HMI"."Screen no by function")
   END_RUNG
   // the same network as SCL:
   "R_TRIG_DB_23"(CLK := "Functions"."2k"."regeration program selected", Q => "HMI"."Function ONS".regeneration);   // R_TRIG
   IF "Functions"."2k"."regeration program selected" AND "HMI"."Function ONS".regeneration THEN
       "HMI"."Current screen No" := 1014;
   END_IF;
   IF "Functions"."2k"."regeration program selected" THEN "HMI"."Screen no by function" := 1014; END_IF;
END_REGION

REGION Network 18: Main menu
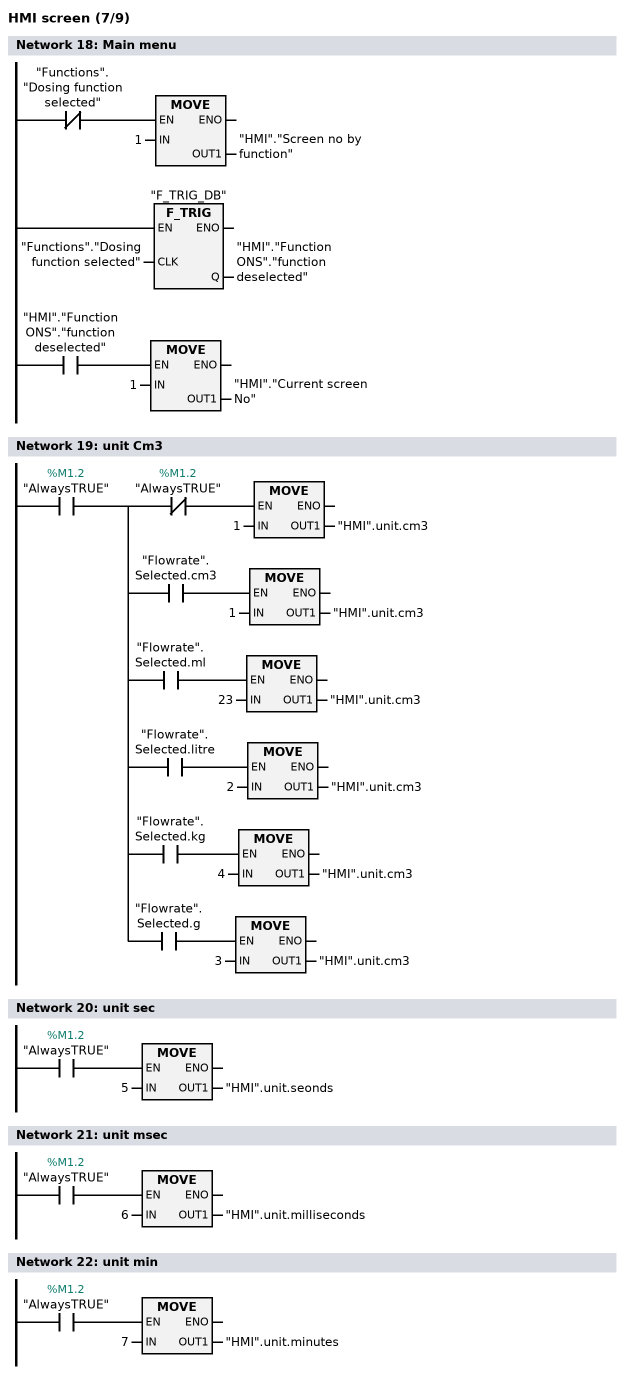
   RUNG wire#powerrail
      I_Contact( "Functions"."Dosing function selected" )
      Move(in := 1, out1 => "HMI"."Screen no by function")
   END_RUNG
   RUNG wire#powerrail
      "F_TRIG_DB".F_TRIG(CLK := "Functions"."Dosing function selected", Q => "HMI"."Function ONS"."function deselected")
   END_RUNG
   RUNG wire#powerrail
      Contact( "HMI"."Function ONS"."function deselected" )
      Move(in := 1, out1 => "HMI"."Current screen No")
   END_RUNG
   // the same network as SCL:
   IF NOT "Functions"."Dosing function selected" THEN "HMI"."Screen no by function" := 1; END_IF;
   "F_TRIG_DB"(CLK := "Functions"."Dosing function selected", Q => "HMI"."Function ONS"."function deselected");   // F_TRIG
   IF "HMI"."Function ONS"."function deselected" THEN "HMI"."Current screen No" := 1; END_IF;
END_REGION

REGION Network 19: unit Cm3
   RUNG wire#powerrail
      Contact( "AlwaysTRUE" )
      wire#w1
      I_Contact( "AlwaysTRUE" )
      Move(in := 1, out1 => "HMI".unit.cm3)
   END_RUNG
   RUNG wire#w1
      Contact( "Flowrate".Selected.cm3 )
      Move(in := 1, out1 => "HMI".unit.cm3)
   END_RUNG
   RUNG wire#w1
      Contact( "Flowrate".Selected.ml )
      Move(in := 23, out1 => "HMI".unit.cm3)
   END_RUNG
   RUNG wire#w1
      Contact( "Flowrate".Selected.litre )
      Move(in := 2, out1 => "HMI".unit.cm3)
   END_RUNG
   RUNG wire#w1
      Contact( "Flowrate".Selected.kg )
      Move(in := 4, out1 => "HMI".unit.cm3)
   END_RUNG
   RUNG wire#w1
      Contact( "Flowrate".Selected.g )
      Move(in := 3, out1 => "HMI".unit.cm3)
   END_RUNG
   // the same network as SCL:
   IF "AlwaysTRUE" AND NOT "AlwaysTRUE" THEN "HMI".unit.cm3 := 1; END_IF;
   IF "AlwaysTRUE" AND "Flowrate".Selected.cm3 THEN "HMI".unit.cm3 := 1; END_IF;
   IF "AlwaysTRUE" AND "Flowrate".Selected.ml THEN "HMI".unit.cm3 := 23; END_IF;
   IF "AlwaysTRUE" AND "Flowrate".Selected.litre THEN "HMI".unit.cm3 := 2; END_IF;
   IF "AlwaysTRUE" AND "Flowrate".Selected.kg THEN "HMI".unit.cm3 := 4; END_IF;
   IF "AlwaysTRUE" AND "Flowrate".Selected.g THEN "HMI".unit.cm3 := 3; END_IF;
END_REGION

REGION Network 20: unit sec
   RUNG wire#powerrail
      Contact( "AlwaysTRUE" )
      Move(in := 5, out1 => "HMI".unit.seonds)
   END_RUNG
   // the same network as SCL:
   IF "AlwaysTRUE" THEN "HMI".unit.seonds := 5; END_IF;
END_REGION

REGION Network 21: unit msec
   RUNG wire#powerrail
      Contact( "AlwaysTRUE" )
      Move(in := 6, out1 => "HMI".unit.milliseconds)
   END_RUNG
   // the same network as SCL:
   IF "AlwaysTRUE" THEN "HMI".unit.milliseconds := 6; END_IF;
END_REGION

REGION Network 22: unit min
   RUNG wire#powerrail
      Contact( "AlwaysTRUE" )
      Move(in := 7, out1 => "HMI".unit.minutes)
   END_RUNG
   // the same network as SCL:
   IF "AlwaysTRUE" THEN "HMI".unit.minutes := 7; END_IF;
END_REGION

REGION Network 23: unit hour
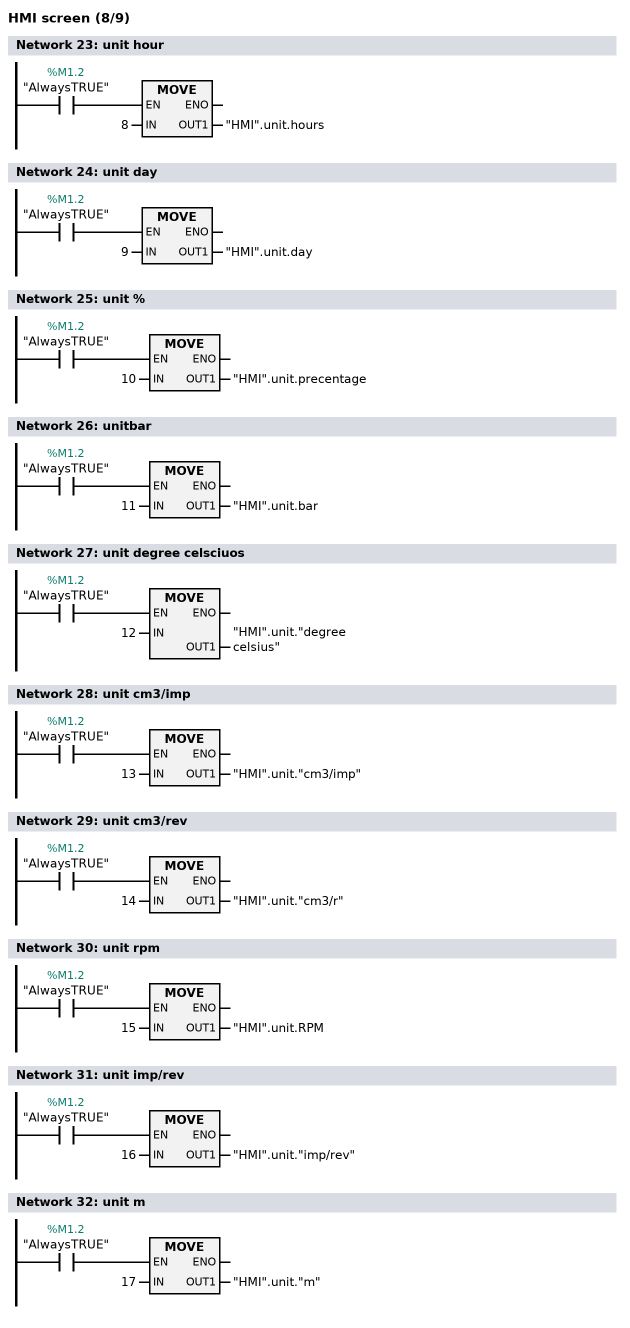
   RUNG wire#powerrail
      Contact( "AlwaysTRUE" )
      Move(in := 8, out1 => "HMI".unit.hours)
   END_RUNG
   // the same network as SCL:
   IF "AlwaysTRUE" THEN "HMI".unit.hours := 8; END_IF;
END_REGION

REGION Network 24: unit day
   RUNG wire#powerrail
      Contact( "AlwaysTRUE" )
      Move(in := 9, out1 => "HMI".unit.day)
   END_RUNG
   // the same network as SCL:
   IF "AlwaysTRUE" THEN "HMI".unit.day := 9; END_IF;
END_REGION

REGION Network 25: unit %
   RUNG wire#powerrail
      Contact( "AlwaysTRUE" )
      Move(in := 10, out1 => "HMI".unit.precentage)
   END_RUNG
   // the same network as SCL:
   IF "AlwaysTRUE" THEN "HMI".unit.precentage := 10; END_IF;
END_REGION

REGION Network 26: unitbar
   RUNG wire#powerrail
      Contact( "AlwaysTRUE" )
      Move(in := 11, out1 => "HMI".unit.bar)
   END_RUNG
   // the same network as SCL:
   IF "AlwaysTRUE" THEN "HMI".unit.bar := 11; END_IF;
END_REGION

REGION Network 27: unit degree celsciuos
   RUNG wire#powerrail
      Contact( "AlwaysTRUE" )
      Move(in := 12, out1 => "HMI".unit."degree celsius")
   END_RUNG
   // the same network as SCL:
   IF "AlwaysTRUE" THEN "HMI".unit."degree celsius" := 12; END_IF;
END_REGION

REGION Network 28: unit cm3/imp
   RUNG wire#powerrail
      Contact( "AlwaysTRUE" )
      Move(in := 13, out1 => "HMI".unit."cm3/imp")
   END_RUNG
   // the same network as SCL:
   IF "AlwaysTRUE" THEN "HMI".unit."cm3/imp" := 13; END_IF;
END_REGION

REGION Network 29: unit cm3/rev
   RUNG wire#powerrail
      Contact( "AlwaysTRUE" )
      Move(in := 14, out1 => "HMI".unit."cm3/r")
   END_RUNG
   // the same network as SCL:
   IF "AlwaysTRUE" THEN "HMI".unit."cm3/r" := 14; END_IF;
END_REGION

REGION Network 30: unit rpm
   RUNG wire#powerrail
      Contact( "AlwaysTRUE" )
      Move(in := 15, out1 => "HMI".unit.RPM)
   END_RUNG
   // the same network as SCL:
   IF "AlwaysTRUE" THEN "HMI".unit.RPM := 15; END_IF;
END_REGION

REGION Network 31: unit imp/rev
   RUNG wire#powerrail
      Contact( "AlwaysTRUE" )
      Move(in := 16, out1 => "HMI".unit."imp/rev")
   END_RUNG
   // the same network as SCL:
   IF "AlwaysTRUE" THEN "HMI".unit."imp/rev" := 16; END_IF;
END_REGION

REGION Network 32: unit m
   RUNG wire#powerrail
      Contact( "AlwaysTRUE" )
      Move(in := 17, out1 => "HMI".unit."m")
   END_RUNG
   // the same network as SCL:
   IF "AlwaysTRUE" THEN "HMI".unit."m" := 17; END_IF;
END_REGION

REGION Network 33: unit cm3/min
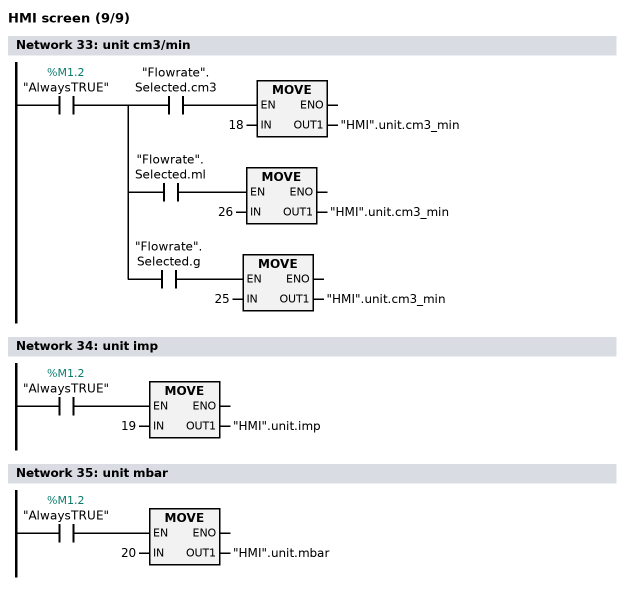
   RUNG wire#powerrail
      Contact( "AlwaysTRUE" )
      wire#w1
      Contact( "Flowrate".Selected.cm3 )
      Move(in := 18, out1 => "HMI".unit.cm3_min)
   END_RUNG
   RUNG wire#w1
      Contact( "Flowrate".Selected.ml )
      Move(in := 26, out1 => "HMI".unit.cm3_min)
   END_RUNG
   RUNG wire#w1
      Contact( "Flowrate".Selected.g )
      Move(in := 25, out1 => "HMI".unit.cm3_min)
   END_RUNG
   // the same network as SCL:
   IF "AlwaysTRUE" AND "Flowrate".Selected.cm3 THEN "HMI".unit.cm3_min := 18; END_IF;
   IF "AlwaysTRUE" AND "Flowrate".Selected.ml THEN "HMI".unit.cm3_min := 26; END_IF;
   IF "AlwaysTRUE" AND "Flowrate".Selected.g THEN "HMI".unit.cm3_min := 25; END_IF;
END_REGION

REGION Network 34: unit imp
   RUNG wire#powerrail
      Contact( "AlwaysTRUE" )
      Move(in := 19, out1 => "HMI".unit.imp)
   END_RUNG
   // the same network as SCL:
   IF "AlwaysTRUE" THEN "HMI".unit.imp := 19; END_IF;
END_REGION

REGION Network 35: unit mbar
   RUNG wire#powerrail
      Contact( "AlwaysTRUE" )
      Move(in := 20, out1 => "HMI".unit.mbar)
   END_RUNG
   // the same network as SCL:
   IF "AlwaysTRUE" THEN "HMI".unit.mbar := 20; END_IF;
END_REGION

REGION Network 36 (SCL): user logged
   IF "HMI"."HMI User" = WString#'admin' THEN
       "HMI".AdminLogged := true;

   ELSE
       "HMI".AdminLogged := false;
       "HMI".userlogged := FALSE;
   END_IF;


   IF LEN("HMI"."HMI User") > 1 THEN
       "HMI".userlogged := TRUE;
   ELSE
       "HMI".userlogged := FALSE;
   END_IF;
END_REGION

REGION Network 37 (SCL)
   "HMI"."HMI user To hmi" := "HMI"."HMI User";
END_REGION
END_FUNCTION

FUNCTION "Flowrate adjustment configuration A" : Void   // FC9, LAD
{ S7_Optimized_Access := 'TRUE' }
VERSION : 0.1
// stored: AutoNumber true, IsIECCheckEnabled false, SetENOAutomatically false, UDAEnableTagReadback false
BEGIN

REGION Network 1 (SCL)
   IF "Pump & Flowrate"."Calculated flowrate A without adjustment" <= "Pump & Flowrate".capacity."Pump A" * 0.05 THEN
       "Pump & Flowrate"."fowrate A Adjustment Configuration" := "Flowrate adjustment A".percentage."5%";
   ELSIF "Pump & Flowrate"."Calculated flowrate A without adjustment" <= "Pump & Flowrate".capacity."Pump A" * 0.10 THEN
       "Pump & Flowrate"."fowrate A Adjustment Configuration" := "Flowrate adjustment A".percentage."10%";
   ELSIF "Pump & Flowrate"."Calculated flowrate A without adjustment" <= "Pump & Flowrate".capacity."Pump A" * 0.15 THEN
       "Pump & Flowrate"."fowrate A Adjustment Configuration" := "Flowrate adjustment A".percentage."15%";
   ELSIF "Pump & Flowrate"."Calculated flowrate A without adjustment" <= "Pump & Flowrate".capacity."Pump A" * 0.20 THEN
       "Pump & Flowrate"."fowrate A Adjustment Configuration" := "Flowrate adjustment A".percentage."20%";
   ELSIF "Pump & Flowrate"."Calculated flowrate A without adjustment" <= "Pump & Flowrate".capacity."Pump A" * 0.25 THEN
       "Pump & Flowrate"."fowrate A Adjustment Configuration" := "Flowrate adjustment A".percentage."25%";
   ELSIF "Pump & Flowrate"."Calculated flowrate A without adjustment" <= "Pump & Flowrate".capacity."Pump A" * 0.30 THEN
       "Pump & Flowrate"."fowrate A Adjustment Configuration" := "Flowrate adjustment A".percentage."30%";
   ELSIF "Pump & Flowrate"."Calculated flowrate A without adjustment" <= "Pump & Flowrate".capacity."Pump A" * 0.40 THEN
       "Pump & Flowrate"."fowrate A Adjustment Configuration" := "Flowrate adjustment A".percentage."40%";
   ELSIF "Pump & Flowrate"."Calculated flowrate A without adjustment" <= "Pump & Flowrate".capacity."Pump A" * 0.50 THEN
       "Pump & Flowrate"."fowrate A Adjustment Configuration" := "Flowrate adjustment A".percentage."50%";
   ELSIF "Pump & Flowrate"."Calculated flowrate A without adjustment" <= "Pump & Flowrate".capacity."Pump A" * 0.60 THEN
       "Pump & Flowrate"."fowrate A Adjustment Configuration" := "Flowrate adjustment A".percentage."60%";
   ELSIF "Pump & Flowrate"."Calculated flowrate A without adjustment" <= "Pump & Flowrate".capacity."Pump A" * 0.70 THEN
       "Pump & Flowrate"."fowrate A Adjustment Configuration" := "Flowrate adjustment A".percentage."70%";
   ELSIF "Pump & Flowrate"."Calculated flowrate A without adjustment" <= "Pump & Flowrate".capacity."Pump A" * 0.80 THEN
       "Pump & Flowrate"."fowrate A Adjustment Configuration" := "Flowrate adjustment A".percentage."80%";
   ELSIF "Pump & Flowrate"."Calculated flowrate A without adjustment" <= "Pump & Flowrate".capacity."Pump A" * 0.90 THEN
       "Pump & Flowrate"."fowrate A Adjustment Configuration" := "Flowrate adjustment A".percentage."90%";
   ELSE
       "Pump & Flowrate"."fowrate A Adjustment Configuration" := "Flowrate adjustment A".percentage."100%";
   END_IF;
END_REGION

REGION Network 3: reset alladjustment
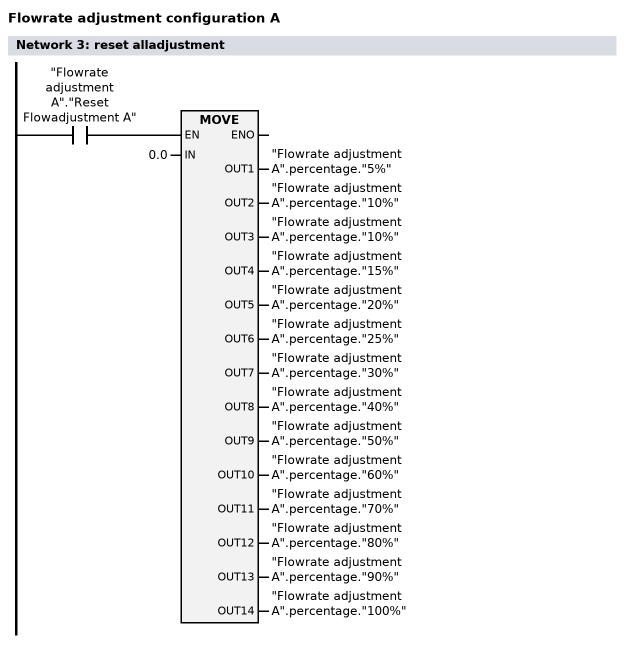
   RUNG wire#powerrail
      Contact( "Flowrate adjustment A"."Reset Flowadjustment A" )
      Move(in := 0.0, out1 => "Flowrate adjustment A".percentage."5%", out2 => "Flowrate adjustment A".percentage."10%", out3 => "Flowrate adjustment A".percentage."10%", out4 => "Flowrate adjustment A".percentage."15%", out5 => "Flowrate adjustment A".percentage."20%", out6 => "Flowrate adjustment A".percentage."25%", out7 => "Flowrate adjustment A".percentage."30%", out8 => "Flowrate adjustment A".percentage."40%", out9 => "Flowrate adjustment A".percentage."50%", out10 => "Flowrate adjustment A".percentage."60%", out11 => "Flowrate adjustment A".percentage."70%", out12 => "Flowrate adjustment A".percentage."80%", out13 => "Flowrate adjustment A".percentage."90%", out14 => "Flowrate adjustment A".percentage."100%")
   END_RUNG
   // the same network as SCL:
   IF "Flowrate adjustment A"."Reset Flowadjustment A" THEN
       "Flowrate adjustment A".percentage."5%" := 0.0;
       "Flowrate adjustment A".percentage."10%" := 0.0;
       "Flowrate adjustment A".percentage."10%" := 0.0;
       "Flowrate adjustment A".percentage."15%" := 0.0;
       "Flowrate adjustment A".percentage."20%" := 0.0;
       "Flowrate adjustment A".percentage."25%" := 0.0;
       "Flowrate adjustment A".percentage."30%" := 0.0;
       "Flowrate adjustment A".percentage."40%" := 0.0;
       "Flowrate adjustment A".percentage."50%" := 0.0;
       "Flowrate adjustment A".percentage."60%" := 0.0;
       "Flowrate adjustment A".percentage."70%" := 0.0;
       "Flowrate adjustment A".percentage."80%" := 0.0;
       "Flowrate adjustment A".percentage."90%" := 0.0;
       "Flowrate adjustment A".percentage."100%" := 0.0;
   END_IF;
END_REGION
END_FUNCTION

FUNCTION "Flowrate adjustment configuration B" : Void   // FC10, LAD
{ S7_Optimized_Access := 'TRUE' }
VERSION : 0.1
// stored: AutoNumber false, IsIECCheckEnabled false, SetENOAutomatically false, UDAEnableTagReadback false
BEGIN

REGION Network 1 (SCL)
   IF "Pump & Flowrate"."Calculated Flowrate B without adjustment" <= "Pump & Flowrate".capacity."pump B" * 0.05 THEN
       "Pump & Flowrate"."fowrate B Adjustment Configuration" := "Flowrate adjustment B".percentage."5%";
   ELSIF "Pump & Flowrate"."Calculated Flowrate B without adjustment" <= "Pump & Flowrate".capacity."pump B" * 0.10 THEN
       "Pump & Flowrate"."fowrate B Adjustment Configuration" := "Flowrate adjustment B".percentage."10%";
   ELSIF "Pump & Flowrate"."Calculated Flowrate B without adjustment" <= "Pump & Flowrate".capacity."pump B" * 0.15 THEN
       "Pump & Flowrate"."fowrate B Adjustment Configuration" := "Flowrate adjustment B".percentage."15%";
   ELSIF "Pump & Flowrate"."Calculated Flowrate B without adjustment" <= "Pump & Flowrate".capacity."pump B" * 0.20 THEN
       "Pump & Flowrate"."fowrate B Adjustment Configuration" := "Flowrate adjustment B".percentage."20%";
   ELSIF "Pump & Flowrate"."Calculated Flowrate B without adjustment" <= "Pump & Flowrate".capacity."pump B" * 0.25 THEN
       "Pump & Flowrate"."fowrate B Adjustment Configuration" := "Flowrate adjustment B".percentage."25%";
   ELSIF "Pump & Flowrate"."Calculated Flowrate B without adjustment" <= "Pump & Flowrate".capacity."pump B" * 0.30 THEN
       "Pump & Flowrate"."fowrate B Adjustment Configuration" := "Flowrate adjustment B".percentage."30%";
   ELSIF "Pump & Flowrate"."Calculated Flowrate B without adjustment" <= "Pump & Flowrate".capacity."pump B" * 0.40 THEN
       "Pump & Flowrate"."fowrate B Adjustment Configuration" := "Flowrate adjustment B".percentage."40%";
   ELSIF "Pump & Flowrate"."Calculated Flowrate B without adjustment" <= "Pump & Flowrate".capacity."pump B" * 0.50 THEN
       "Pump & Flowrate"."fowrate B Adjustment Configuration" := "Flowrate adjustment B".percentage."50%";
   ELSIF "Pump & Flowrate"."Calculated Flowrate B without adjustment" <= "Pump & Flowrate".capacity."pump B" * 0.60 THEN
       "Pump & Flowrate"."fowrate B Adjustment Configuration" := "Flowrate adjustment B".percentage."60%";
   ELSIF "Pump & Flowrate"."Calculated Flowrate B without adjustment" <= "Pump & Flowrate".capacity."pump B" * 0.70 THEN
       "Pump & Flowrate"."fowrate B Adjustment Configuration" := "Flowrate adjustment B".percentage."70%";
   ELSIF "Pump & Flowrate"."Calculated Flowrate B without adjustment" <= "Pump & Flowrate".capacity."pump B" * 0.80 THEN
       "Pump & Flowrate"."fowrate B Adjustment Configuration" := "Flowrate adjustment B".percentage."80%";
   ELSIF "Pump & Flowrate"."Calculated Flowrate B without adjustment" <= "Pump & Flowrate".capacity."pump B" * 0.90 THEN
       "Pump & Flowrate"."fowrate B Adjustment Configuration" := "Flowrate adjustment B".percentage."90%";
   ELSE
       "Pump & Flowrate"."fowrate B Adjustment Configuration" := "Flowrate adjustment B".percentage."100%";
   END_IF;
END_REGION

REGION Network 2: reset alladjustment
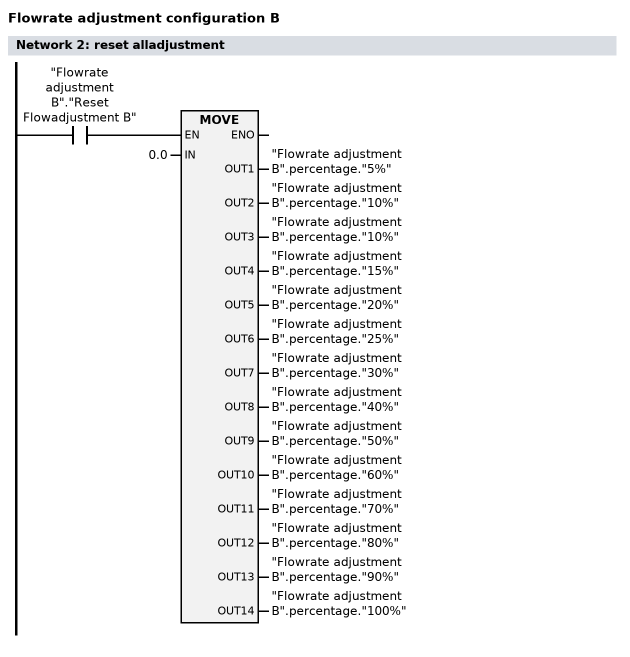
   RUNG wire#powerrail
      Contact( "Flowrate adjustment B"."Reset Flowadjustment B" )
      Move(in := 0.0, out1 => "Flowrate adjustment B".percentage."5%", out2 => "Flowrate adjustment B".percentage."10%", out3 => "Flowrate adjustment B".percentage."10%", out4 => "Flowrate adjustment B".percentage."15%", out5 => "Flowrate adjustment B".percentage."20%", out6 => "Flowrate adjustment B".percentage."25%", out7 => "Flowrate adjustment B".percentage."30%", out8 => "Flowrate adjustment B".percentage."40%", out9 => "Flowrate adjustment B".percentage."50%", out10 => "Flowrate adjustment B".percentage."60%", out11 => "Flowrate adjustment B".percentage."70%", out12 => "Flowrate adjustment B".percentage."80%", out13 => "Flowrate adjustment B".percentage."90%", out14 => "Flowrate adjustment B".percentage."100%")
   END_RUNG
   // the same network as SCL:
   IF "Flowrate adjustment B"."Reset Flowadjustment B" THEN
       "Flowrate adjustment B".percentage."5%" := 0.0;
       "Flowrate adjustment B".percentage."10%" := 0.0;
       "Flowrate adjustment B".percentage."10%" := 0.0;
       "Flowrate adjustment B".percentage."15%" := 0.0;
       "Flowrate adjustment B".percentage."20%" := 0.0;
       "Flowrate adjustment B".percentage."25%" := 0.0;
       "Flowrate adjustment B".percentage."30%" := 0.0;
       "Flowrate adjustment B".percentage."40%" := 0.0;
       "Flowrate adjustment B".percentage."50%" := 0.0;
       "Flowrate adjustment B".percentage."60%" := 0.0;
       "Flowrate adjustment B".percentage."70%" := 0.0;
       "Flowrate adjustment B".percentage."80%" := 0.0;
       "Flowrate adjustment B".percentage."90%" := 0.0;
       "Flowrate adjustment B".percentage."100%" := 0.0;
   END_IF;
END_REGION
END_FUNCTION

FUNCTION "Function & start signal" : Void   // FC3, LAD
{ S7_Optimized_Access := 'TRUE' }
VERSION : 0.1
// stored: AutoNumber true, IsIECCheckEnabled false, SetENOAutomatically false, UDAEnableTagReadback false
   VAR_TEMP   // added for the SCL form of the ladder/FBD networks
      _w1 : Bool;
      _w2 : Bool;
      _w3 : Bool;
   END_VAR
BEGIN

REGION Network 1: Move dearing A Flowrate to Main register
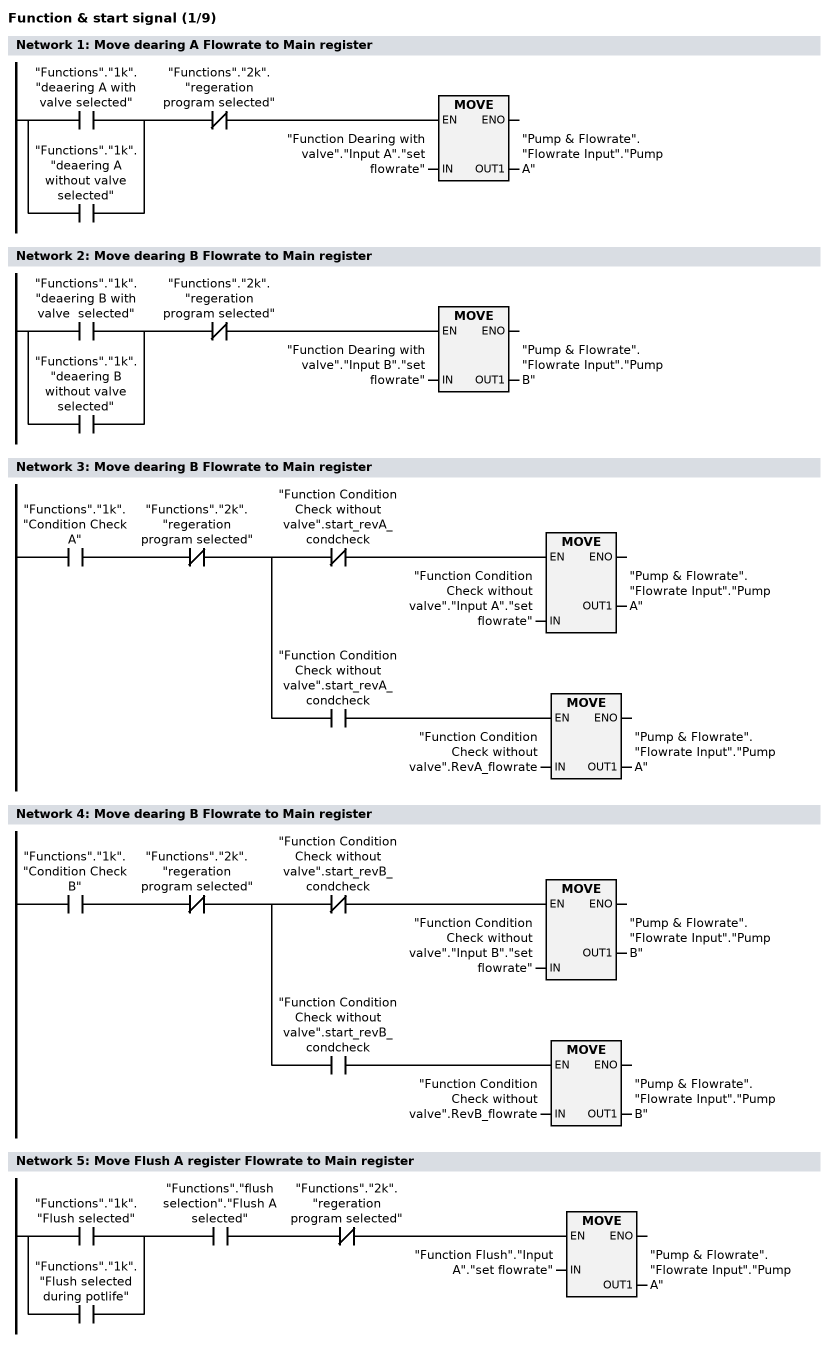
   IF ("Functions"."1k"."deaering A with valve selected" OR "Functions"."1k"."deaering A without valve selected") AND NOT "Functions"."2k"."regeration program selected" THEN
       "Pump & Flowrate"."Flowrate Input"."Pump A" := "Function Dearing with valve"."Input A"."set flowrate";
   END_IF;
END_REGION

REGION Network 2: Move dearing B Flowrate to Main register
   IF ("Functions"."1k"."deaering B with valve  selected" OR "Functions"."1k"."deaering B without valve  selected") AND NOT "Functions"."2k"."regeration program selected" THEN
       "Pump & Flowrate"."Flowrate Input"."Pump B" := "Function Dearing with valve"."Input B"."set flowrate";
   END_IF;
END_REGION

REGION Network 3: Move dearing B Flowrate to Main register
   #_w1 := "Functions"."1k"."Condition Check A" AND NOT "Functions"."2k"."regeration program selected";
   IF #_w1 AND NOT "Function ConditionCheck without valve".start_revA_condcheck THEN
       "Pump & Flowrate"."Flowrate Input"."Pump A" := "Function ConditionCheck without valve"."Input A"."set flowrate";
   END_IF;
   IF #_w1 AND "Function ConditionCheck without valve".start_revA_condcheck THEN
       "Pump & Flowrate"."Flowrate Input"."Pump A" := "Function ConditionCheck without valve".RevA_flowrate;
   END_IF;
END_REGION

REGION Network 4: Move dearing B Flowrate to Main register
   #_w1 := "Functions"."1k"."Condition Check B" AND NOT "Functions"."2k"."regeration program selected";
   IF #_w1 AND NOT "Function ConditionCheck without valve".start_revB_condcheck THEN
       "Pump & Flowrate"."Flowrate Input"."Pump B" := "Function ConditionCheck without valve"."Input B"."set flowrate";
   END_IF;
   IF #_w1 AND "Function ConditionCheck without valve".start_revB_condcheck THEN
       "Pump & Flowrate"."Flowrate Input"."Pump B" := "Function ConditionCheck without valve".RevB_flowrate;
   END_IF;
END_REGION

REGION Network 5: Move Flush A register Flowrate to Main register
   IF ("Functions"."1k"."Flush selected" OR "Functions"."1k"."Flush selected during potlife") AND "Functions"."flush selection"."Flush A selected" AND NOT "Functions"."2k"."regeration program selected" THEN
       "Pump & Flowrate"."Flowrate Input"."Pump A" := "Function Flush"."Input A"."set flowrate";
   END_IF;
END_REGION

REGION Network 6: Move Flush B register Flowrate to Main register
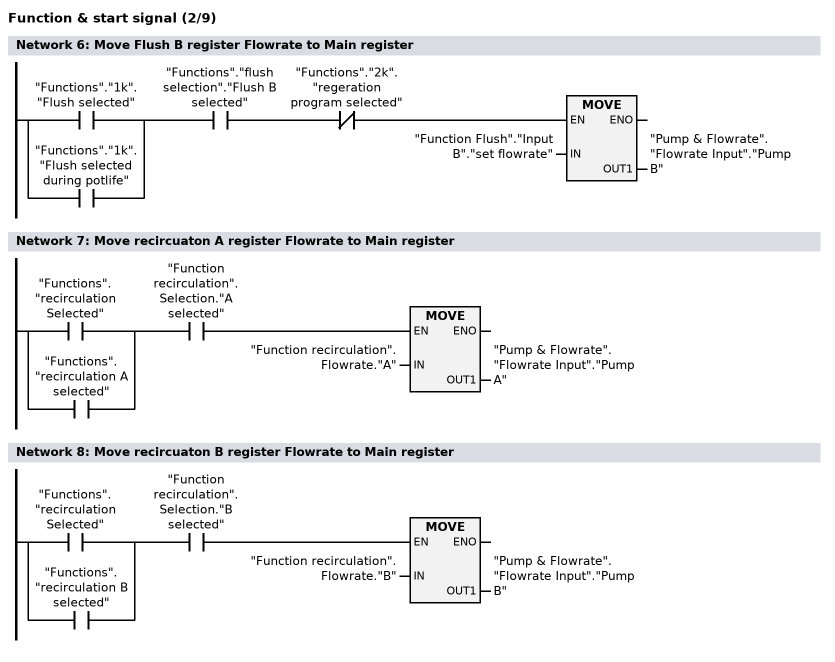
   IF ("Functions"."1k"."Flush selected" OR "Functions"."1k"."Flush selected during potlife") AND "Functions"."flush selection"."Flush B selected" AND NOT "Functions"."2k"."regeration program selected" THEN
       "Pump & Flowrate"."Flowrate Input"."Pump B" := "Function Flush"."Input B"."set flowrate";
   END_IF;
END_REGION

REGION Network 7: Move recircuaton A register Flowrate to Main register
   IF ("Functions"."recirculation Selected" OR "Functions"."recirculation A selected") AND "Function recirculation".Selection."A selected" THEN
       "Pump & Flowrate"."Flowrate Input"."Pump A" := "Function recirculation".Flowrate."A";
   END_IF;
END_REGION

REGION Network 8: Move recircuaton B register Flowrate to Main register
   IF ("Functions"."recirculation Selected" OR "Functions"."recirculation B selected") AND "Function recirculation".Selection."B selected" THEN
       "Pump & Flowrate"."Flowrate Input"."Pump B" := "Function recirculation".Flowrate."B";
   END_IF;
END_REGION

REGION Network 9: Move Metering program register Flowrate to Main register
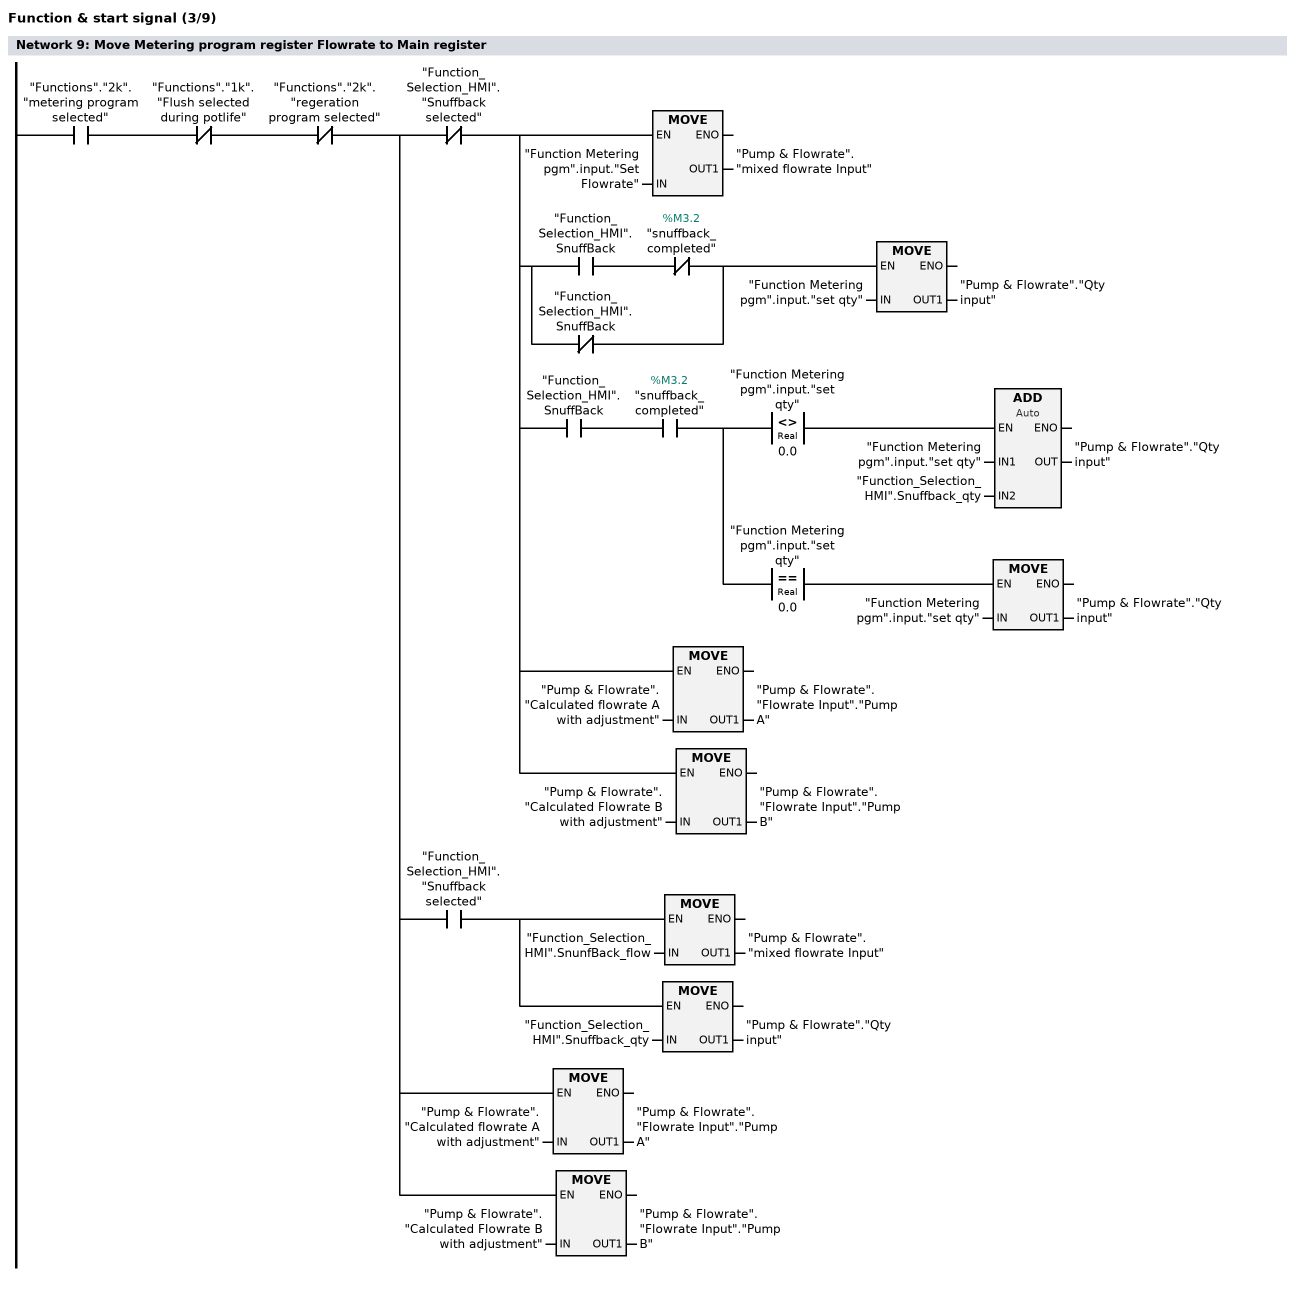
   #_w1 := "Functions"."2k"."metering program selected" AND NOT "Functions"."1k"."Flush selected during potlife" AND NOT "Functions"."2k"."regeration program selected";
   #_w2 := #_w1 AND NOT "Function_Selection_HMI"."Snuffback selected";
   IF #_w2 THEN
       "Pump & Flowrate"."mixed flowrate Input" := "Function Metering pgm".input."Set Flowrate";
   END_IF;
   IF #_w2 AND (("Function_Selection_HMI".SnuffBack AND NOT "snuffback_completed") OR NOT "Function_Selection_HMI".SnuffBack) THEN
       "Pump & Flowrate"."Qty input" := "Function Metering pgm".input."set qty";
   END_IF;
   #_w3 := #_w2 AND "Function_Selection_HMI".SnuffBack AND "snuffback_completed";
   IF #_w3 AND ("Function Metering pgm".input."set qty" <> 0.0) THEN
       "Pump & Flowrate"."Qty input" := "Function Metering pgm".input."set qty" + "Function_Selection_HMI".Snuffback_qty;
   END_IF;
   IF #_w3 AND ("Function Metering pgm".input."set qty" = 0.0) THEN
       "Pump & Flowrate"."Qty input" := "Function Metering pgm".input."set qty";
   END_IF;
   IF #_w2 THEN
       "Pump & Flowrate"."Flowrate Input"."Pump A" := "Pump & Flowrate"."Calculated flowrate A with adjustment";
       "Pump & Flowrate"."Flowrate Input"."Pump B" := "Pump & Flowrate"."Calculated Flowrate B  with adjustment";
   END_IF;
   IF #_w1 AND "Function_Selection_HMI"."Snuffback selected" THEN
       "Pump & Flowrate"."mixed flowrate Input" := "Function_Selection_HMI".SnunfBack_flow;
       "Pump & Flowrate"."Qty input" := "Function_Selection_HMI".Snuffback_qty;
   END_IF;
   IF #_w1 THEN
       "Pump & Flowrate"."Flowrate Input"."Pump A" := "Pump & Flowrate"."Calculated flowrate A with adjustment";
       "Pump & Flowrate"."Flowrate Input"."Pump B" := "Pump & Flowrate"."Calculated Flowrate B  with adjustment";
   END_IF;
END_REGION

REGION Network 10: Move shot Metering register Flowrate to Main register
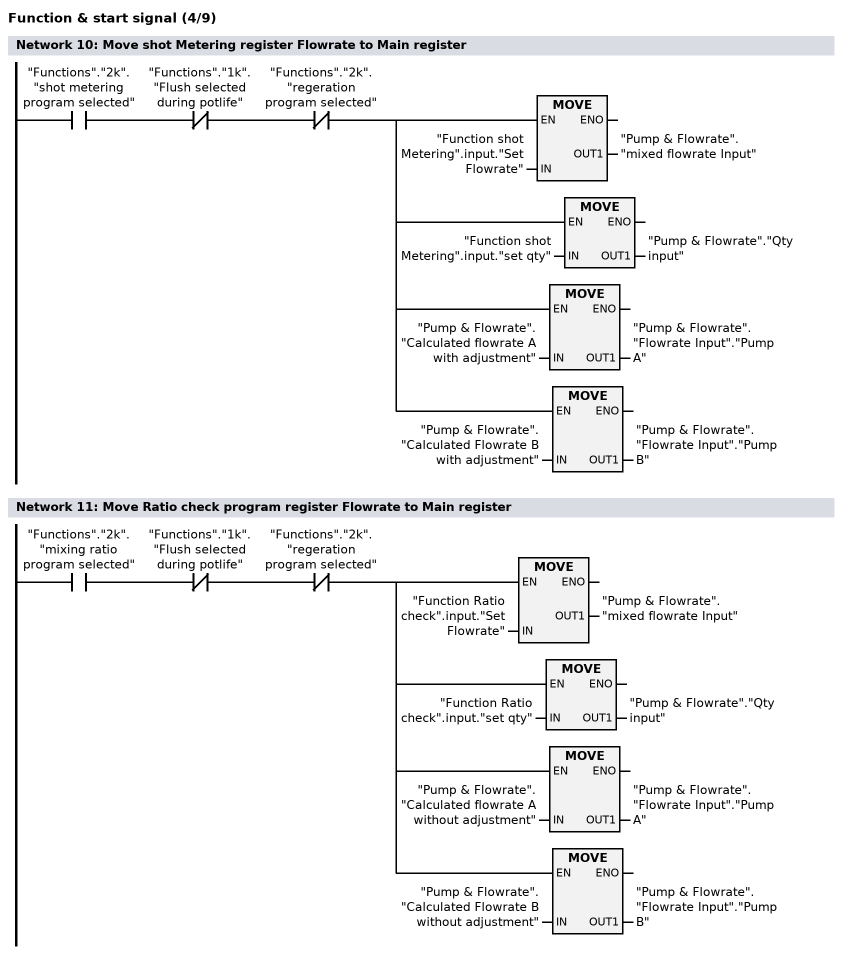
   IF "Functions"."2k"."shot metering program selected" AND NOT "Functions"."1k"."Flush selected during potlife" AND NOT "Functions"."2k"."regeration program selected" THEN
       "Pump & Flowrate"."mixed flowrate Input" := "Function shot Metering".input."Set Flowrate";
       "Pump & Flowrate"."Qty input" := "Function shot Metering".input."set qty";
       "Pump & Flowrate"."Flowrate Input"."Pump A" := "Pump & Flowrate"."Calculated flowrate A with adjustment";
       "Pump & Flowrate"."Flowrate Input"."Pump B" := "Pump & Flowrate"."Calculated Flowrate B  with adjustment";
   END_IF;
END_REGION

REGION Network 11: Move Ratio check program register Flowrate to Main register
   IF "Functions"."2k"."mixing ratio program selected" AND NOT "Functions"."1k"."Flush selected during potlife" AND NOT "Functions"."2k"."regeration program selected" THEN
       "Pump & Flowrate"."mixed flowrate Input" := "Function Ratio check".input."Set Flowrate";
       "Pump & Flowrate"."Qty input" := "Function Ratio check".input."set qty";
       "Pump & Flowrate"."Flowrate Input"."Pump A" := "Pump & Flowrate"."Calculated flowrate A without adjustment";
       "Pump & Flowrate"."Flowrate Input"."Pump B" := "Pump & Flowrate"."Calculated Flowrate B without adjustment";
   END_IF;
END_REGION

REGION Network 12: Move Pre run program register Flowrate to Main register
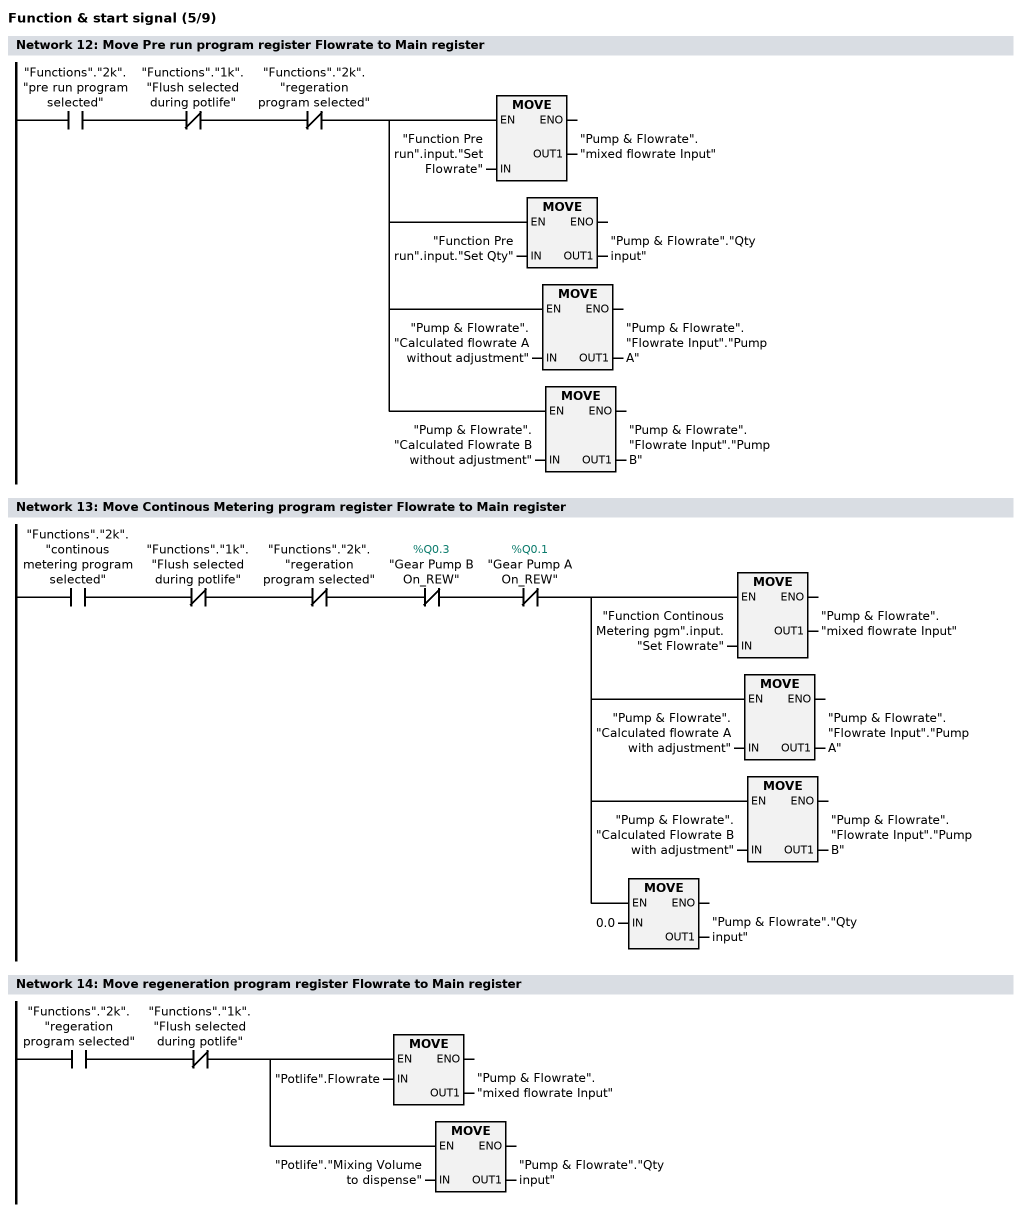
   IF "Functions"."2k"."pre run program selected" AND NOT "Functions"."1k"."Flush selected during potlife" AND NOT "Functions"."2k"."regeration program selected" THEN
       "Pump & Flowrate"."mixed flowrate Input" := "Function Pre run".input."Set Flowrate";
       "Pump & Flowrate"."Qty input" := "Function Pre run".input."Set Qty";
       "Pump & Flowrate"."Flowrate Input"."Pump A" := "Pump & Flowrate"."Calculated flowrate A without adjustment";
       "Pump & Flowrate"."Flowrate Input"."Pump B" := "Pump & Flowrate"."Calculated Flowrate B without adjustment";
   END_IF;
END_REGION

REGION Network 13: Move Continous Metering program register Flowrate to Main register
   IF "Functions"."2k"."continous metering program selected" AND NOT "Functions"."1k"."Flush selected during potlife" AND NOT "Functions"."2k"."regeration program selected" AND NOT "Gear Pump B On_REW" AND NOT "Gear Pump A On_REW" THEN
       "Pump & Flowrate"."mixed flowrate Input" := "Function Continous Metering pgm".input."Set Flowrate";
       "Pump & Flowrate"."Flowrate Input"."Pump A" := "Pump & Flowrate"."Calculated flowrate A with adjustment";
       "Pump & Flowrate"."Flowrate Input"."Pump B" := "Pump & Flowrate"."Calculated Flowrate B  with adjustment";
       "Pump & Flowrate"."Qty input" := 0.0;
   END_IF;
END_REGION

REGION Network 14: Move regeneration program register Flowrate to Main register
   IF "Functions"."2k"."regeration program selected" AND NOT "Functions"."1k"."Flush selected during potlife" THEN
       "Pump & Flowrate"."mixed flowrate Input" := "Potlife".Flowrate;
       "Pump & Flowrate"."Qty input" := "Potlife"."Mixing Volume to dispense";
   END_IF;
END_REGION

REGION Network 15: Dearing with valve A start/stop
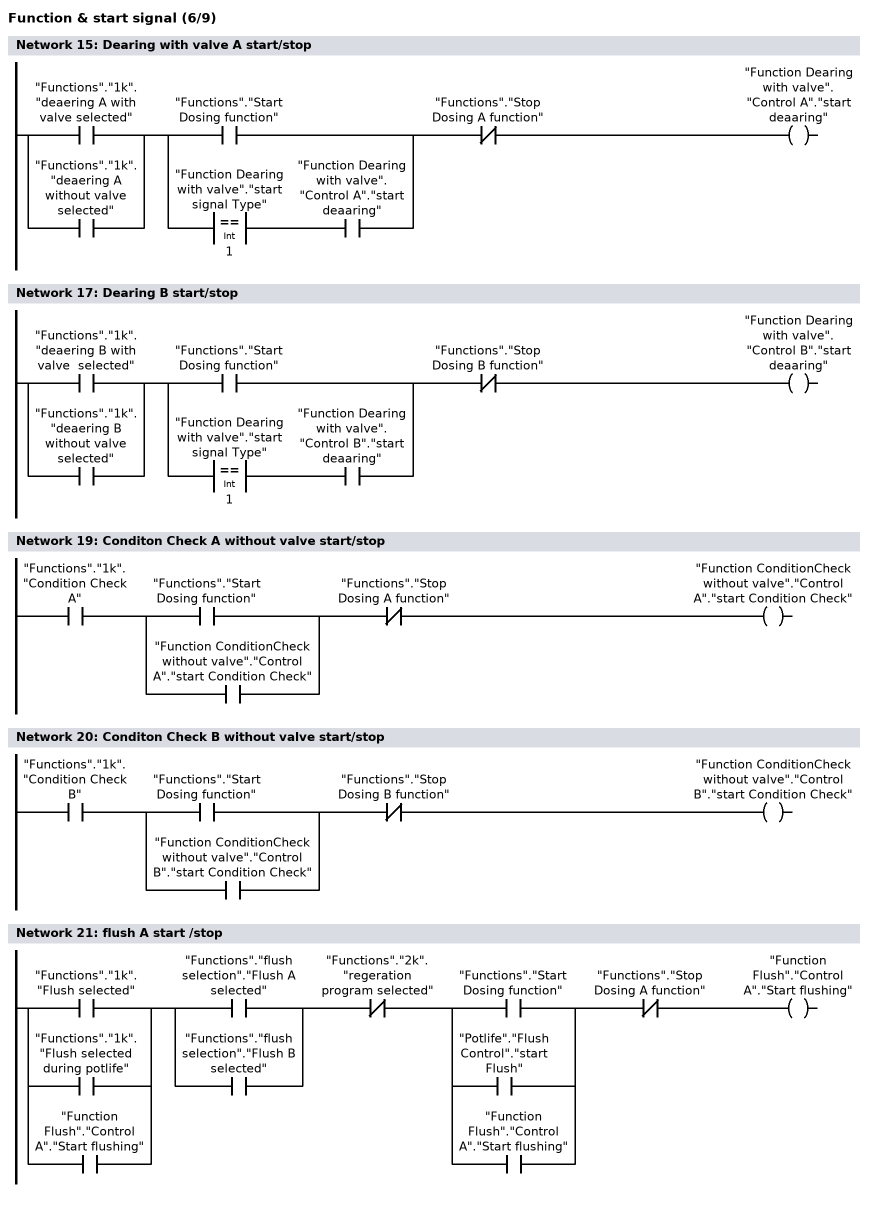
   RUNG wire#powerrail
      Contact( "Functions"."1k"."deaering A with valve selected" )
      wire#w1
      Contact( "Functions"."Start Dosing function" )
      wire#w2
      I_Contact( "Functions"."Stop Dosing A function" )
      Coil( "Function Dearing with valve"."Control A"."start deaaring" )
   END_RUNG
   RUNG wire#powerrail
      Contact( "Functions"."1k"."deaering A without valve selected" )
   END_RUNG wire#w1
   RUNG wire#w1
      { S7_Templates := "SrcType := Int" } EQ_Contact(in1 := "Function Dearing with valve"."start signal Type", in2 := 1)
      Contact( "Function Dearing with valve"."Control A"."start deaaring" )
   END_RUNG wire#w2
   // the same network as SCL:
   "Function Dearing with valve"."Control A"."start deaaring" := ("Functions"."1k"."deaering A with valve selected" OR "Functions"."1k"."deaering A without valve selected") AND ("Functions"."Start Dosing function" OR (("Function Dearing with valve"."start signal Type" = 1) AND "Function Dearing with valve"."Control A"."start deaaring")) AND NOT "Functions"."Stop Dosing A function";
END_REGION

REGION Network 16: Dearing without valve A start/stop
END_REGION

REGION Network 17: Dearing B start/stop
   RUNG wire#powerrail
      Contact( "Functions"."1k"."deaering B with valve  selected" )
      wire#w1
      Contact( "Functions"."Start Dosing function" )
      wire#w2
      I_Contact( "Functions"."Stop Dosing B function" )
      Coil( "Function Dearing with valve"."Control B"."start deaaring" )
   END_RUNG
   RUNG wire#powerrail
      Contact( "Functions"."1k"."deaering B without valve  selected" )
   END_RUNG wire#w1
   RUNG wire#w1
      { S7_Templates := "SrcType := Int" } EQ_Contact(in1 := "Function Dearing with valve"."start signal Type", in2 := 1)
      Contact( "Function Dearing with valve"."Control B"."start deaaring" )
   END_RUNG wire#w2
   // the same network as SCL:
   "Function Dearing with valve"."Control B"."start deaaring" := ("Functions"."1k"."deaering B with valve  selected" OR "Functions"."1k"."deaering B without valve  selected") AND ("Functions"."Start Dosing function" OR (("Function Dearing with valve"."start signal Type" = 1) AND "Function Dearing with valve"."Control B"."start deaaring")) AND NOT "Functions"."Stop Dosing B function";
END_REGION

REGION Network 18: Dearing B without valve start/stop
END_REGION

REGION Network 19: Conditon Check A without valve start/stop
   RUNG wire#powerrail
      Contact( "Functions"."1k"."Condition Check A" )
      wire#w1
      Contact( "Functions"."Start Dosing function" )
      wire#w2
      I_Contact( "Functions"."Stop Dosing A function" )
      Coil( "Function ConditionCheck without valve"."Control A"."start Condition Check" )
   END_RUNG
   RUNG wire#w1
      Contact( "Function ConditionCheck without valve"."Control A"."start Condition Check" )
   END_RUNG wire#w2
   // the same network as SCL:
   "Function ConditionCheck without valve"."Control A"."start Condition Check" := "Functions"."1k"."Condition Check A" AND ("Functions"."Start Dosing function" OR "Function ConditionCheck without valve"."Control A"."start Condition Check") AND NOT "Functions"."Stop Dosing A function";
END_REGION

REGION Network 20: Conditon Check B without valve start/stop
   RUNG wire#powerrail
      Contact( "Functions"."1k"."Condition Check B" )
      wire#w1
      Contact( "Functions"."Start Dosing function" )
      wire#w2
      I_Contact( "Functions"."Stop Dosing B function" )
      Coil( "Function ConditionCheck without valve"."Control B"."start Condition Check" )
   END_RUNG
   RUNG wire#w1
      Contact( "Function ConditionCheck without valve"."Control B"."start Condition Check" )
   END_RUNG wire#w2
   // the same network as SCL:
   "Function ConditionCheck without valve"."Control B"."start Condition Check" := "Functions"."1k"."Condition Check B" AND ("Functions"."Start Dosing function" OR "Function ConditionCheck without valve"."Control B"."start Condition Check") AND NOT "Functions"."Stop Dosing B function";
END_REGION

REGION Network 21: flush A start /stop
   RUNG wire#powerrail
      Contact( "Functions"."1k"."Flush selected" )
      wire#w1
      Contact( "Functions"."flush selection"."Flush A selected" )
      wire#w2
      I_Contact( "Functions"."2k"."regeration program selected" )
      wire#w3
      Contact( "Functions"."Start Dosing function" )
      wire#w4
      I_Contact( "Functions"."Stop Dosing A function" )
      Coil( "Function Flush"."Control A"."Start flushing" )
   END_RUNG
   RUNG wire#powerrail
      Contact( "Functions"."1k"."Flush selected during potlife" )
   END_RUNG wire#w1
   RUNG wire#powerrail
      Contact( "Function Flush"."Control A"."Start flushing" )
   END_RUNG wire#w1
   RUNG wire#w1
      Contact( "Functions"."flush selection"."Flush B selected" )
   END_RUNG wire#w2
   RUNG wire#w3
      Contact( "Potlife"."Flush Control"."start Flush" )
   END_RUNG wire#w4
   RUNG wire#w3
      Contact( "Function Flush"."Control A"."Start flushing" )
   END_RUNG wire#w4
   // the same network as SCL:
   "Function Flush"."Control A"."Start flushing" := ("Functions"."1k"."Flush selected" OR "Functions"."1k"."Flush selected during potlife" OR "Function Flush"."Control A"."Start flushing") AND ("Functions"."flush selection"."Flush A selected" OR "Functions"."flush selection"."Flush B selected") AND NOT "Functions"."2k"."regeration program selected" AND ("Functions"."Start Dosing function" OR "Potlife"."Flush Control"."start Flush" OR "Function Flush"."Control A"."Start flushing") AND NOT "Functions"."Stop Dosing A function";
END_REGION

REGION Network 22: flush B start /stop
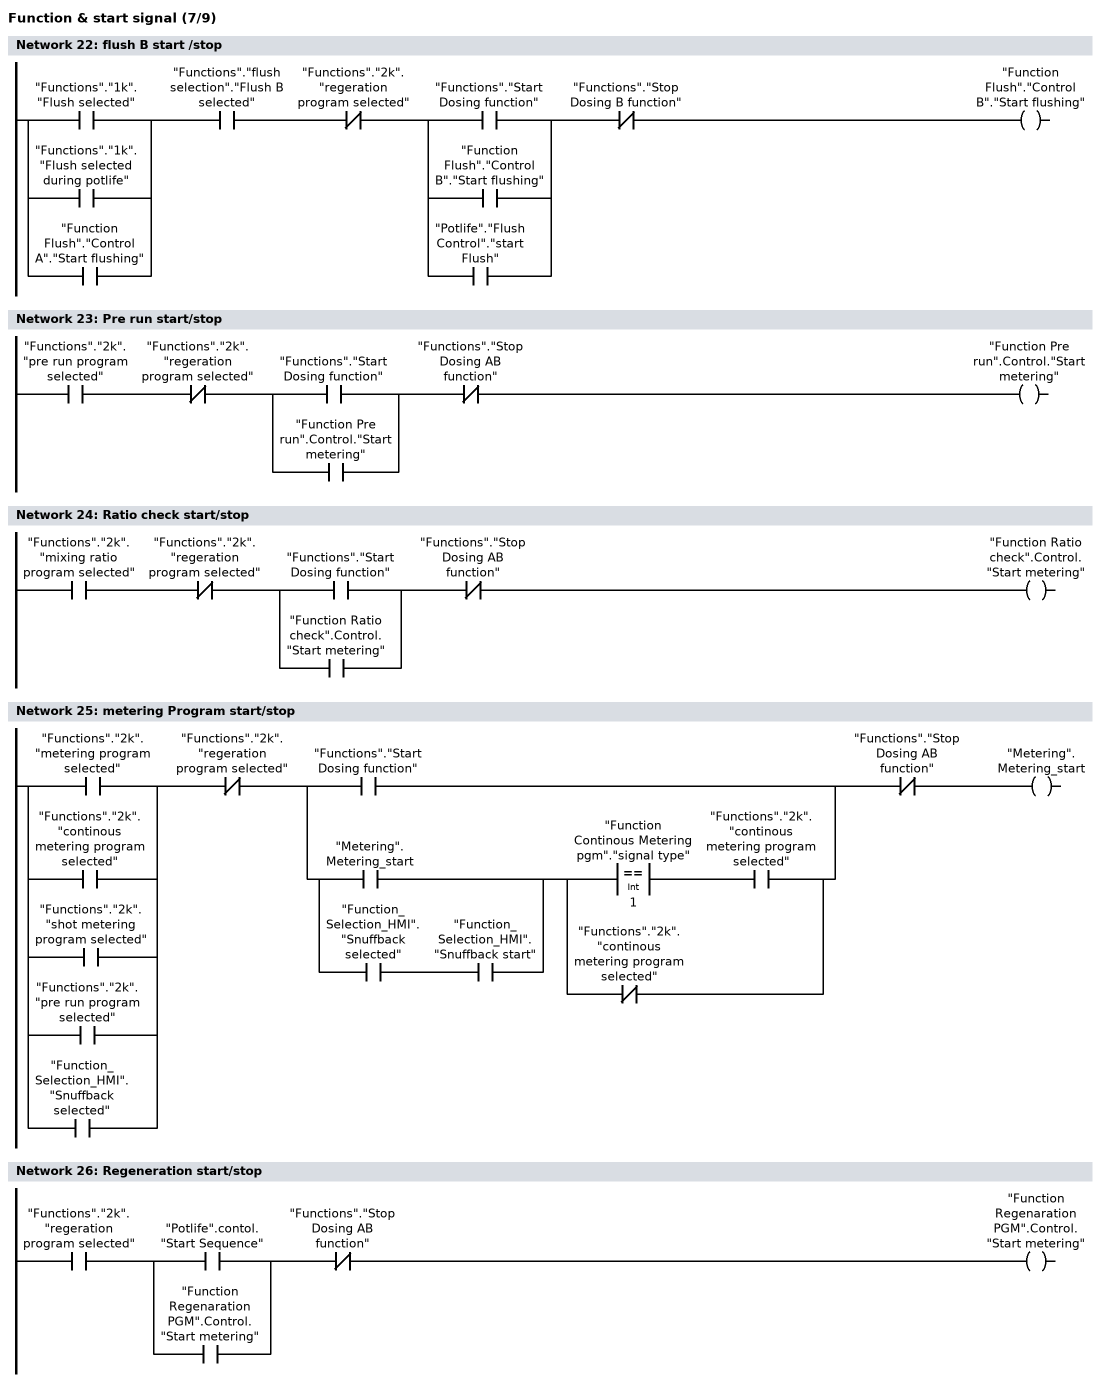
   RUNG wire#powerrail
      Contact( "Functions"."1k"."Flush selected" )
      wire#w1
      Contact( "Functions"."flush selection"."Flush B selected" )
      I_Contact( "Functions"."2k"."regeration program selected" )
      wire#w2
      Contact( "Functions"."Start Dosing function" )
      wire#w3
      I_Contact( "Functions"."Stop Dosing B function" )
      Coil( "Function Flush"."Control B"."Start flushing" )
   END_RUNG
   RUNG wire#powerrail
      Contact( "Functions"."1k"."Flush selected during potlife" )
   END_RUNG wire#w1
   RUNG wire#powerrail
      Contact( "Function Flush"."Control A"."Start flushing" )
   END_RUNG wire#w1
   RUNG wire#w2
      Contact( "Function Flush"."Control B"."Start flushing" )
   END_RUNG wire#w3
   RUNG wire#w2
      Contact( "Potlife"."Flush Control"."start Flush" )
   END_RUNG wire#w3
   // the same network as SCL:
   "Function Flush"."Control B"."Start flushing" := ("Functions"."1k"."Flush selected" OR "Functions"."1k"."Flush selected during potlife" OR "Function Flush"."Control A"."Start flushing") AND "Functions"."flush selection"."Flush B selected" AND NOT "Functions"."2k"."regeration program selected" AND ("Functions"."Start Dosing function" OR "Function Flush"."Control B"."Start flushing" OR "Potlife"."Flush Control"."start Flush") AND NOT "Functions"."Stop Dosing B function";
END_REGION

REGION Network 23: Pre run start/stop
   RUNG wire#powerrail
      Contact( "Functions"."2k"."pre run program selected" )
      I_Contact( "Functions"."2k"."regeration program selected" )
      wire#w1
      Contact( "Functions"."Start Dosing function" )
      wire#w2
      I_Contact( "Functions"."Stop Dosing AB function" )
      Coil( "Function Pre run".Control."Start metering" )
   END_RUNG
   RUNG wire#w1
      Contact( "Function Pre run".Control."Start metering" )
   END_RUNG wire#w2
   // the same network as SCL:
   "Function Pre run".Control."Start metering" := "Functions"."2k"."pre run program selected" AND NOT "Functions"."2k"."regeration program selected" AND ("Functions"."Start Dosing function" OR "Function Pre run".Control."Start metering") AND NOT "Functions"."Stop Dosing AB function";
END_REGION

REGION Network 24: Ratio check start/stop
   RUNG wire#powerrail
      Contact( "Functions"."2k"."mixing ratio program selected" )
      I_Contact( "Functions"."2k"."regeration program selected" )
      wire#w1
      Contact( "Functions"."Start Dosing function" )
      wire#w2
      I_Contact( "Functions"."Stop Dosing AB function" )
      Coil( "Function Ratio check".Control."Start metering" )
   END_RUNG
   RUNG wire#w1
      Contact( "Function Ratio check".Control."Start metering" )
   END_RUNG wire#w2
   // the same network as SCL:
   "Function Ratio check".Control."Start metering" := "Functions"."2k"."mixing ratio program selected" AND NOT "Functions"."2k"."regeration program selected" AND ("Functions"."Start Dosing function" OR "Function Ratio check".Control."Start metering") AND NOT "Functions"."Stop Dosing AB function";
END_REGION

REGION Network 25: metering Program start/stop
   RUNG wire#powerrail
      Contact( "Functions"."2k"."metering program selected" )
      wire#w1
      I_Contact( "Functions"."2k"."regeration program selected" )
      wire#w2
      Contact( "Functions"."Start Dosing function" )
      wire#w3
      I_Contact( "Functions"."Stop Dosing AB function" )
      Coil( "Metering".Metering_start )
   END_RUNG
   RUNG wire#powerrail
      Contact( "Functions"."2k"."continous metering program selected" )
   END_RUNG wire#w1
   RUNG wire#powerrail
      Contact( "Functions"."2k"."shot metering program selected" )
   END_RUNG wire#w1
   RUNG wire#powerrail
      Contact( "Functions"."2k"."pre run program selected" )
   END_RUNG wire#w1
   RUNG wire#powerrail
      Contact( "Function_Selection_HMI"."Snuffback selected" )
   END_RUNG wire#w1
   RUNG wire#w2
      Contact( "Metering".Metering_start )
      wire#w4
      { S7_Templates := "SrcType := Int" } EQ_Contact(in1 := "Function Continous Metering pgm"."signal type", in2 := 1)
      Contact( "Functions"."2k"."continous metering program selected" )
   END_RUNG wire#w3
   RUNG wire#w2
      Contact( "Function_Selection_HMI"."Snuffback selected" )
      Contact( "Function_Selection_HMI"."Snuffback start" )
   END_RUNG wire#w4
   RUNG wire#w4
      I_Contact( "Functions"."2k"."continous metering program selected" )
   END_RUNG wire#w3
   // the same network as SCL:
   "Metering".Metering_start := ("Functions"."2k"."metering program selected" OR "Functions"."2k"."continous metering program selected" OR "Functions"."2k"."shot metering program selected" OR "Functions"."2k"."pre run program selected" OR "Function_Selection_HMI"."Snuffback selected") AND NOT "Functions"."2k"."regeration program selected" AND ("Functions"."Start Dosing function" OR (("Metering".Metering_start OR ("Function_Selection_HMI"."Snuffback selected" AND "Function_Selection_HMI"."Snuffback start")) AND ((("Function Continous Metering pgm"."signal type" = 1) AND "Functions"."2k"."continous metering program selected") OR NOT "Functions"."2k"."continous metering program selected"))) AND NOT "Functions"."Stop Dosing AB function";
END_REGION

REGION Network 26: Regeneration start/stop
   RUNG wire#powerrail
      Contact( "Functions"."2k"."regeration program selected" )
      wire#w1
      Contact( "Potlife".contol."Start Sequence" )
      wire#w2
      I_Contact( "Functions"."Stop Dosing AB function" )
      Coil( "Function Regenaration PGM".Control."Start metering" )
   END_RUNG
   RUNG wire#w1
      Contact( "Function Regenaration PGM".Control."Start metering" )
   END_RUNG wire#w2
   // the same network as SCL:
   "Function Regenaration PGM".Control."Start metering" := "Functions"."2k"."regeration program selected" AND ("Potlife".contol."Start Sequence" OR "Function Regenaration PGM".Control."Start metering") AND NOT "Functions"."Stop Dosing AB function";
END_REGION

REGION Network 27: metering Shot start/stop
